LIN {X 0,Y 509.461,Z 538.867,A -85,B 0,C 180,E1 -5497.53,E2 -5497.53} C_VEL
LIN {X 0,Y 509.618,Z 532.772,A -85,B 0,C 180,E1 -5498.525,E2 -5498.525} C_VEL
LIN {X 0,Y 509.848,Z 525.444,A -85,B 0,C 180,E1 -5499.521,E2 -5499.521} C_VEL
LIN {X 0,Y 510.009,Z 518.515,A -85,B 0,C 180,E1 -5500.32,E2 -5500.32} C_VEL
LIN {X 0,Y 510.319,Z 510.334,A -85,B 0,C 180,E1 -5501.116,E2 -5501.116} C_VEL
LIN {X 0,Y 510.583,Z 501.821,A -85,B 0,C 180,E1 -5501.815,E2 -5501.815} C_VEL
LIN {X 0,Y 510.841,Z 492.093,A -85,B 0,C 180,E1 -5502.475,E2 -5502.475} C_VEL
LIN {X 0,Y 511.112,Z 482.332,A -85,B 0,C 180,E1 -5503.012,E2 -5503.012} C_VEL
LIN {X 0,Y 511.344,Z 473.256,A -85,B 0,C 180,E1 -5503.411,E2 -5503.411} C_VEL
LIN {X 0,Y 511.519,Z 463.74,A -85,B 0,C 180,E1 -5503.735,E2 -5503.735} C_VEL
LIN {X 0,Y 511.764,Z 453.432,A -85,B 0,C 180,E1 -5503.981,E2 -5503.981} C_VEL
LIN {X 0,Y 512.128,Z 381.828,A -85,B 0,C 180,E1 -5505.012,E2 -5505.012} C_VEL
LIN {X 0,Y 512.114,Z 359.712,A -85,B 0,C 180,E1 -5505.327,E2 -5505.327} C_VEL
LIN {X 0,Y 510.045,Z 347.334,A -85,B 0,C 180,E1 -5505.59,E2 -5505.59} C_VEL
LIN {X 0,Y 510.232,Z 339.032,A -85,B 0,C 180,E1 -5507.226,E2 -5507.226} C_VEL
LIN {X 0,Y 510.588,Z 324.426,A -85,B 0,C 180,E1 -5510.127,E2 -5510.127} C_VEL
LIN {X 0,Y 510.987,Z 310.909,A -85,B 0,C 180,E1 -5512.852,E2 -5512.852} C_VEL
LIN {X 0,Y 511.208,Z 302.536,A -85,B 0,C 180,E1 -5514.592,E2 -5514.592} C_VEL
LIN {X 0,Y 509.916,Z 294.495,A -85,B 0,C 180,E1 -5516.407,E2 -5516.407} C_VEL
LIN {X 0,Y 509.872,Z 294.473,A -85,B 0,C 180,E1 -5518.844,E2 -5518.844} C_VEL
LIN {X 0,Y 509.82,Z 294.481,A -85,B 0,C 180,E1 -5521.589,E2 -5521.589} C_VEL
LIN {X 0,Y 509.845,Z 294.474,A -85,B 0,C 180,E1 -5524.413,E2 -5524.413} C_VEL
LIN {X 0,Y 509.806,Z 294.478,A -85,B 0,C 180,E1 -5527.341,E2 -5527.341} C_VEL
LIN {X 0,Y 509.835,Z 294.468,A -85,B 0,C 180,E1 -5530.381,E2 -5530.381} C_VEL
LIN {X 0,Y 509.819,Z 294.476,A -85,B 0,C 180,E1 -5533.061,E2 -5533.061} C_VEL
LIN {X 0,Y 509.818,Z 294.48,A -85,B 0,C 180,E1 -5535.792,E2 -5535.792} C_VEL
LIN {X 0,Y 509.854,Z 294.47,A -85,B 0,C 180,E1 -5538.574,E2 -5538.574} C_VEL
LIN {X 0,Y 509.845,Z 294.479,A -85,B 0,C 180,E1 -5541.786,E2 -5541.786} C_VEL
LIN {X 0,Y 509.824,Z 294.472,A -85,B 0,C 180,E1 -5544.621,E2 -5544.621} C_VEL
LIN {X 0,Y 509.853,Z 294.472,A -85,B 0,C 180,E1 -5547.48,E2 -5547.48} C_VEL
LIN {X 0,Y 509.852,Z 294.471,A -85,B 0,C 180,E1 -5550.273,E2 -5550.273} C_VEL
LIN {X 0,Y 509.878,Z 294.462,A -85,B 0,C 180,E1 -5552.944,E2 -5552.944} C_VEL
LIN {X 0,Y 509.839,Z 294.478,A -85,B 0,C 180,E1 -5555.572,E2 -5555.572} C_VEL
LIN {X 0,Y 509.814,Z 294.475,A -85,B 0,C 180,E1 -5558.148,E2 -5558.148} C_VEL
LIN {X 0,Y 509.856,Z 294.463,A -85,B 0,C 180,E1 -5560.681,E2 -5560.681} C_VEL
LIN {X 0,Y 509.876,Z 294.465,A -85,B 0,C 180,E1 -5563.174,E2 -5563.174} C_VEL
LIN {X 0,Y 509.865,Z 294.474,A -85,B 0,C 180,E1 -5565.634,E2 -5565.634} C_VEL
LIN {X 0,Y 509.908,Z 294.462,A -85,B 0,C 180,E1 -5568.874,E2 -5568.874} C_VEL
LIN {X 0,Y 509.943,Z 294.455,A -85,B 0,C 180,E1 -5572.078,E2 -5572.078} C_VEL
LIN {X 0,Y 509.973,Z 294.455,A -85,B 0,C 180,E1 -5574.464,E2 -5574.464} C_VEL
LIN {X 0,Y 510.043,Z 294.446,A -85,B 0,C 180,E1 -5577.63,E2 -5577.63} C_VEL
LIN {X 0,Y 510.043,Z 294.435,A -85,B 0,C 180,E1 -5580,E2 -5580} C_VEL
LIN {X 0,Y 510.044,Z 294.442,A -85,B 0,C 180,E1 -5582.369,E2 -5582.369} C_VEL
LIN {X 0,Y 509.967,Z 294.456,A -85,B 0,C 180,E1 -5586.329,E2 -5586.329} C_VEL
LIN {X 0,Y 509.906,Z 294.463,A -85,B 0,C 180,E1 -5588.72,E2 -5588.72} C_VEL
LIN {X 0,Y 509.895,Z 294.462,A -85,B 0,C 180,E1 -5591.931,E2 -5591.931} C_VEL
LIN {X 0,Y 509.883,Z 294.472,A -85,B 0,C 180,E1 -5595.242,E2 -5595.242} C_VEL
LIN {X 0,Y 509.877,Z 294.462,A -85,B 0,C 180,E1 -5598.001,E2 -5598.001} C_VEL
LIN {X 0,Y 509.84,Z 294.475,A -85,B 0,C 180,E1 -5601.002,E2 -5601.002} C_VEL
LIN {X 0,Y 509.859,Z 294.473,A -85,B 0,C 180,E1 -5604.426,E2 -5604.426} C_VEL
LIN {X 0,Y 509.875,Z 294.466,A -85,B 0,C 180,E1 -5607.056,E2 -5607.056} C_VEL
LIN {X 0,Y 509.871,Z 294.468,A -85,B 0,C 180,E1 -5609.75,E2 -5609.75} C_VEL
LIN {X 0,Y 509.867,Z 294.474,A -85,B 0,C 180,E1 -5612.775,E2 -5612.775} C_VEL
LIN {X 0,Y 509.833,Z 294.471,A -85,B 0,C 180,E1 -5615.581,E2 -5615.581} C_VEL
LIN {X 0,Y 509.843,Z 294.477,A -85,B 0,C 180,E1 -5618.338,E2 -5618.338} C_VEL
LIN {X 0,Y 509.856,Z 294.469,A -85,B 0,C 180,E1 -5621.425,E2 -5621.425} C_VEL
LIN {X 0,Y 509.848,Z 294.476,A -85,B 0,C 180,E1 -5624.668,E2 -5624.668} C_VEL
LIN {X 0,Y 509.853,Z 294.459,A -85,B 0,C 180,E1 -5628.103,E2 -5628.103} C_VEL
LIN {X 0,Y 509.84,Z 294.478,A -85,B 0,C 180,E1 -5630.648,E2 -5630.648} C_VEL
LIN {X 0,Y 509.824,Z 294.473,A -85,B 0,C 180,E1 -5633.749,E2 -5633.749} C_VEL
LIN {X 0,Y 509.159,Z 294.557,A -85,B 0,C 180,E1 -5634.409,E2 -5634.409} C_VEL
LIN {X 0,Y 506.341,Z 294.908,A -85,B 0,C 180,E1 -5635.481,E2 -5635.481} C_VEL
LIN {X 0,Y 503.947,Z 295.208,A -85,B 0,C 180,E1 -5636.344,E2 -5636.344} C_VEL
LIN {X 0,Y 502.899,Z 295.34,A -85,B 0,C 180,E1 -5637.011,E2 -5637.011} C_VEL
LIN {X 0,Y 502.802,Z 295.35,A -85,B 0,C 180,E1 -5637.236,E2 -5637.236} C_VEL
LIN {X 0,Y 502.809,Z 295.351,A -85,B 0,C 180,E1 -5640.065,E2 -5640.065} C_VEL
LIN {X 0,Y 502.83,Z 295.353,A -85,B 0,C 180,E1 -5642.534,E2 -5642.534} C_VEL
LIN {X 0,Y 502.824,Z 295.348,A -85,B 0,C 180,E1 -5645.299,E2 -5645.299} C_VEL
LIN {X 0,Y 502.78,Z 295.356,A -85,B 0,C 180,E1 -5647.827,E2 -5647.827} C_VEL
LIN {X 0,Y 502.822,Z 295.355,A -85,B 0,C 180,E1 -5650.401,E2 -5650.401} C_VEL
LIN {X 0,Y 502.831,Z 295.349,A -85,B 0,C 180,E1 -5652.932,E2 -5652.932} C_VEL
LIN {X 0,Y 502.841,Z 295.347,A -85,B 0,C 180,E1 -5655.429,E2 -5655.429} C_VEL
LIN {X 0,Y 502.874,Z 295.345,A -85,B 0,C 180,E1 -5658.717,E2 -5658.717} C_VEL
LIN {X 0,Y 502.898,Z 295.345,A -85,B 0,C 180,E1 -5661.967,E2 -5661.967} C_VEL
LIN {X 0,Y 502.936,Z 295.339,A -85,B 0,C 180,E1 -5664.387,E2 -5664.387} C_VEL
LIN {X 0,Y 503.023,Z 295.327,A -85,B 0,C 180,E1 -5667.598,E2 -5667.598} C_VEL
LIN {X 0,Y 503.025,Z 295.33,A -85,B 0,C 180,E1 -5670,E2 -5670} C_VEL
LIN {X 0,Y 503.023,Z 295.327,A -85,B 0,C 180,E1 -5672.402,E2 -5672.402} C_VEL
LIN {X 0,Y 502.936,Z 295.339,A -85,B 0,C 180,E1 -5675.613,E2 -5675.613} C_VEL
LIN {X 0,Y 502.898,Z 295.345,A -85,B 0,C 180,E1 -5678.033,E2 -5678.033} C_VEL
LIN {X 0,Y 502.874,Z 295.345,A -85,B 0,C 180,E1 -5681.283,E2 -5681.283} C_VEL
LIN {X 0,Y 502.841,Z 295.347,A -85,B 0,C 180,E1 -5684.571,E2 -5684.571} C_VEL
LIN {X 0,Y 502.858,Z 295.35,A -85,B 0,C 180,E1 -5687.907,E2 -5687.907} C_VEL
LIN {X 0,Y 502.824,Z 295.349,A -85,B 0,C 180,E1 -5690.536,E2 -5690.536} C_VEL
LIN {X 0,Y 502.792,Z 295.354,A -85,B 0,C 180,E1 -5693.04,E2 -5693.04} C_VEL
LIN {X 0,Y 502.837,Z 295.353,A -85,B 0,C 180,E1 -5695.675,E2 -5695.675} C_VEL
LIN {X 0,Y 502.835,Z 295.343,A -85,B 0,C 180,E1 -5698.372,E2 -5698.372} C_VEL
LIN {X 0,Y 502.791,Z 295.358,A -85,B 0,C 180,E1 -5701.499,E2 -5701.499} C_VEL
LIN {X 0,Y 502.8,Z 295.339,A -85,B 0,C 180,E1 -5704.444,E2 -5704.444} C_VEL
LIN {X 0,Y 502.774,Z 295.356,A -85,B 0,C 180,E1 -5707.178,E2 -5707.178} C_VEL
LIN {X 0,Y 502.781,Z 295.347,A -85,B 0,C 180,E1 -5710.015,E2 -5710.015} C_VEL
LIN {X 0,Y 502.795,Z 295.335,A -85,B 0,C 180,E1 -5712.199,E2 -5712.199} C_VEL
LIN {X 0,Y 502.792,Z 295.357,A -85,B 0,C 180,E1 -5715.468,E2 -5715.468} C_VEL
LIN {X 0,Y 502.821,Z 295.347,A -85,B 0,C 180,E1 -5717.864,E2 -5717.864} C_VEL
LIN {X 0,Y 502.801,Z 295.352,A -85,B 0,C 180,E1 -5721.025,E2 -5721.025} C_VEL
LIN {X 0,Y 502.776,Z 295.35,A -85,B 0,C 180,E1 -5724.167,E2 -5724.167} C_VEL
LIN {X 0,Y 502.823,Z 295.348,A -85,B 0,C 180,E1 -5726.993,E2 -5726.993} C_VEL
LIN {X 0,Y 502.821,Z 295.346,A -85,B 0,C 180,E1 -5730.062,E2 -5730.062} C_VEL
LIN {X 0,Y 502.824,Z 295.34,A -85,B 0,C 180,E1 -5732.533,E2 -5732.533} C_VEL
LIN {X 0,Y 502.818,Z 295.353,A -85,B 0,C 180,E1 -5735.298,E2 -5735.298} C_VEL
LIN {X 0,Y 502.783,Z 295.351,A -85,B 0,C 180,E1 -5737.827,E2 -5737.827} C_VEL
LIN {X 0,Y 502.815,Z 295.341,A -85,B 0,C 180,E1 -5740.4,E2 -5740.4} C_VEL
LIN {X 0,Y 502.826,Z 295.348,A -85,B 0,C 180,E1 -5742.932,E2 -5742.932} C_VEL
LIN {X 0,Y 502.834,Z 295.348,A -85,B 0,C 180,E1 -5745.429,E2 -5745.429} C_VEL
LIN {X 0,Y 502.871,Z 295.341,A -85,B 0,C 180,E1 -5748.717,E2 -5748.717} C_VEL
LIN {X 0,Y 502.891,Z 295.333,A -85,B 0,C 180,E1 -5751.967,E2 -5751.967} C_VEL
LIN {X 0,Y 502.928,Z 295.336,A -85,B 0,C 180,E1 -5754.387,E2 -5754.387} C_VEL
LIN {X 0,Y 503.014,Z 295.318,A -85,B 0,C 180,E1 -5757.598,E2 -5757.598} C_VEL
LIN {X 0,Y 503.014,Z 295.309,A -85,B 0,C 180,E1 -5760,E2 -5760} C_VEL
LIN {X 0,Y 503.013,Z 295.322,A -85,B 0,C 180,E1 -5762.403,E2 -5762.403} C_VEL
LIN {X 0,Y 502.929,Z 295.333,A -85,B 0,C 180,E1 -5765.614,E2 -5765.614} C_VEL
LIN {X 0,Y 502.893,Z 295.334,A -85,B 0,C 180,E1 -5768.034,E2 -5768.034} C_VEL
LIN {X 0,Y 502.872,Z 295.337,A -85,B 0,C 180,E1 -5771.284,E2 -5771.284} C_VEL
LIN {X 0,Y 502.843,Z 295.351,A -85,B 0,C 180,E1 -5774.571,E2 -5774.571} C_VEL
LIN {X 0,Y 502.853,Z 295.336,A -85,B 0,C 180,E1 -5777.908,E2 -5777.908} C_VEL
LIN {X 0,Y 502.821,Z 295.349,A -85,B 0,C 180,E1 -5780.537,E2 -5780.537} C_VEL
LIN {X 0,Y 502.781,Z 295.353,A -85,B 0,C 180,E1 -5783.042,E2 -5783.042} C_VEL
LIN {X 0,Y 502.814,Z 295.343,A -85,B 0,C 180,E1 -5785.677,E2 -5785.677} C_VEL
LIN {X 0,Y 502.834,Z 295.347,A -85,B 0,C 180,E1 -5788.373,E2 -5788.373} C_VEL
LIN {X 0,Y 502.786,Z 295.351,A -85,B 0,C 180,E1 -5791.5,E2 -5791.5} C_VEL
LIN {X 0,Y 502.785,Z 295.353,A -85,B 0,C 180,E1 -5794.443,E2 -5794.443} C_VEL
LIN {X 0,Y 502.772,Z 295.353,A -85,B 0,C 180,E1 -5797.179,E2 -5797.179} C_VEL
LIN {X 0,Y 502.783,Z 295.354,A -85,B 0,C 180,E1 -5800.016,E2 -5800.016} C_VEL
LIN {X 0,Y 502.799,Z 295.358,A -85,B 0,C 180,E1 -5802.2,E2 -5802.2} C_VEL
LIN {X 0,Y 502.782,Z 295.352,A -85,B 0,C 180,E1 -5805.471,E2 -5805.471} C_VEL
LIN {X 0,Y 502.792,Z 295.356,A -85,B 0,C 180,E1 -5807.861,E2 -5807.861} C_VEL
LIN {X 0,Y 502.798,Z 295.349,A -85,B 0,C 180,E1 -5811.025,E2 -5811.025} C_VEL
LIN {X 0,Y 502.769,Z 295.354,A -85,B 0,C 180,E1 -5814.171,E2 -5814.171} C_VEL
LIN {X 0,Y 502.832,Z 295.345,A -85,B 0,C 180,E1 -5816.994,E2 -5816.994} C_VEL
LIN {X 0,Y 502.815,Z 295.352,A -85,B 0,C 180,E1 -5820.066,E2 -5820.066} C_VEL
LIN {X 0,Y 502.868,Z 295.346,A -85,B 0,C 180,E1 -5823.211,E2 -5823.211} C_VEL
LIN {X 0,Y 502.924,Z 295.7,A -85,B 0,C 180,E1 -5823.524,E2 -5823.524} C_VEL
LIN {X 0,Y 504.235,Z 303.512,A -85,B 0,C 180,E1 -5825.284,E2 -5825.284} C_VEL
LIN {X 0,Y 503.886,Z 315.919,A -85,B 0,C 180,E1 -5827.878,E2 -5827.878} C_VEL
LIN {X 0,Y 503.426,Z 330.518,A -85,B 0,C 180,E1 -5830.849,E2 -5830.849} C_VEL
LIN {X 0,Y 503.056,Z 344.925,A -85,B 0,C 180,E1 -5833.775,E2 -5833.775} C_VEL
LIN {X 0,Y 503.018,Z 347.127,A -85,B 0,C 180,E1 -5834.185,E2 -5834.185} C_VEL
LIN {X 0,Y 505.389,Z 362.648,A -85,B 0,C 180,E1 -5834.509,E2 -5834.509} C_VEL
LIN {X 0,Y 504.882,Z 451.906,A -85,B 0,C 180,E1 -5835.798,E2 -5835.798} C_VEL
LIN {X 0,Y 504.667,Z 462.672,A -85,B 0,C 180,E1 -5836.049,E2 -5836.049} C_VEL
LIN {X 0,Y 504.48,Z 471.774,A -85,B 0,C 180,E1 -5836.352,E2 -5836.352} C_VEL
LIN {X 0,Y 504.159,Z 482.137,A -85,B 0,C 180,E1 -5836.805,E2 -5836.805} C_VEL
LIN {X 0,Y 503.896,Z 492.03,A -85,B 0,C 180,E1 -5837.358,E2 -5837.358} C_VEL
LIN {X 0,Y 503.667,Z 500.274,A -85,B 0,C 180,E1 -5837.919,E2 -5837.919} C_VEL
LIN {X 0,Y 503.36,Z 509.004,A -85,B 0,C 180,E1 -5838.626,E2 -5838.626} C_VEL
LIN {X 0,Y 503.083,Z 516.401,A -85,B 0,C 180,E1 -5839.333,E2 -5839.333} C_VEL
LIN {X 0,Y 502.851,Z 523.622,A -85,B 0,C 180,E1 -5840.142,E2 -5840.142} C_VEL
LIN {X 0,Y 502.652,Z 529.825,A -85,B 0,C 180,E1 -5840.95,E2 -5840.95} C_VEL
LIN {X 0,Y 502.478,Z 536.362,A -85,B 0,C 180,E1 -5841.96,E2 -5841.96} C_VEL
LIN {X 0,Y 502.328,Z 541.916,A -85,B 0,C 180,E1 -5842.989,E2 -5842.989} C_VEL
LIN {X 0,Y 502.208,Z 546.351,A -85,B 0,C 180,E1 -5843.975,E2 -5843.975} C_VEL
LIN {X 0,Y 502.114,Z 550.671,A -85,B 0,C 180,E1 -5845.183,E2 -5845.183} C_VEL
LIN {X 0,Y 502.139,Z 553.036,A -85,B 0,C 180,E1 -5845.987,E2 -5845.987} C_VEL
LIN {X 0,Y 502.12,Z 554.831,A -85,B 0,C 180,E1 -5846.791,E2 -5846.791} C_VEL
LIN {X 0,Y 502.037,Z 557.269,A -85,B 0,C 180,E1 -5848.396,E2 -5848.396} C_VEL
LIN {X 0,Y 501.991,Z 557.855,A -85,B 0,C 180,E1 -5849.198,E2 -5849.198} C_VEL
LIN {X 0,Y 501.991,Z 557.855,A -85,B 0,C 180,E1 -5850.802,E2 -5850.802} C_VEL
LIN {X 0,Y 502.037,Z 557.269,A -85,B 0,C 180,E1 -5851.604,E2 -5851.604} C_VEL
LIN {X 0,Y 502.12,Z 554.831,A -85,B 0,C 180,E1 -5853.209,E2 -5853.209} C_VEL
LIN {X 0,Y 502.105,Z 551.886,A -85,B 0,C 180,E1 -5854.415,E2 -5854.415} C_VEL
LIN {X 0,Y 502.205,Z 547.904,A -85,B 0,C 180,E1 -5855.622,E2 -5855.622} C_VEL
LIN {X 0,Y 502.27,Z 542.969,A -85,B 0,C 180,E1 -5856.79,E2 -5856.79} C_VEL
LIN {X 0,Y 502.409,Z 537.517,A -85,B 0,C 180,E1 -5857.839,E2 -5857.839} C_VEL
LIN {X 0,Y 502.597,Z 531.2,A -85,B 0,C 180,E1 -5858.848,E2 -5858.848} C_VEL
LIN {X 0,Y 502.807,Z 525.249,A -85,B 0,C 180,E1 -5859.656,E2 -5859.656} C_VEL
LIN {X 0,Y 502.987,Z 518.32,A -85,B 0,C 180,E1 -5860.465,E2 -5860.465} C_VEL
LIN {X 0,Y 503.306,Z 510.139,A -85,B 0,C 180,E1 -5861.273,E2 -5861.273} C_VEL
LIN {X 0,Y 503.602,Z 501.626,A -85,B 0,C 180,E1 -5861.981,E2 -5861.981} C_VEL
LIN {X 0,Y 503.872,Z 492.358,A -85,B 0,C 180,E1 -5862.622,E2 -5862.622} C_VEL
LIN {X 0,Y 504.155,Z 483.145,A -85,B 0,C 180,E1 -5863.144,E2 -5863.144} C_VEL
LIN {X 0,Y 504.445,Z 473.062,A -85,B 0,C 180,E1 -5863.597,E2 -5863.597} C_VEL
LIN {X 0,Y 504.639,Z 463.546,A -85,B 0,C 180,E1 -5863.926,E2 -5863.926} C_VEL
LIN {X 0,Y 504.869,Z 453.238,A -85,B 0,C 180,E1 -5864.176,E2 -5864.176} C_VEL
LIN {X 0,Y 505.244,Z 390.584,A -85,B 0,C 180,E1 -5865.092,E2 -5865.092} C_VEL
LIN {X 0,Y 505.248,Z 360.522,A -85,B 0,C 180,E1 -5865.526,E2 -5865.526} C_VEL
LIN {X 0,Y 503.065,Z 347.271,A -85,B 0,C 180,E1 -5865.804,E2 -5865.804} C_VEL
LIN {X 0,Y 503.028,Z 346.232,A -85,B 0,C 180,E1 -5865.944,E2 -5865.944} C_VEL
LIN {X 0,Y 503.374,Z 332.655,A -85,B 0,C 180,E1 -5868.73,E2 -5868.73} C_VEL
LIN {X 0,Y 503.873,Z 316.967,A -85,B 0,C 180,E1 -5871.907,E2 -5871.907} C_VEL
LIN {X 0,Y 504.263,Z 304.576,A -85,B 0,C 180,E1 -5874.495,E2 -5874.495} C_VEL
LIN {X 0,Y 503.045,Z 296.318,A -85,B 0,C 180,E1 -5876.332,E2 -5876.332} C_VEL
LIN {X 0,Y 502.855,Z 295.361,A -85,B 0,C 180,E1 -5876.622,E2 -5876.622} C_VEL
LIN {X 0,Y 502.822,Z 295.351,A -85,B 0,C 180,E1 -5879.287,E2 -5879.287} C_VEL
LIN {X 0,Y 502.783,Z 295.355,A -85,B 0,C 180,E1 -5882.084,E2 -5882.084} C_VEL
LIN {X 0,Y 502.796,Z 295.35,A -85,B 0,C 180,E1 -5884.965,E2 -5884.965} C_VEL
LIN {X 0,Y 502.791,Z 295.352,A -85,B 0,C 180,E1 -5888.485,E2 -5888.485} C_VEL
LIN {X 0,Y 502.798,Z 295.342,A -85,B 0,C 180,E1 -5891.067,E2 -5891.067} C_VEL
LIN {X 0,Y 502.775,Z 295.354,A -85,B 0,C 180,E1 -5894.339,E2 -5894.339} C_VEL
LIN {X 0,Y 502.768,Z 295.353,A -85,B 0,C 180,E1 -5896.768,E2 -5896.768} C_VEL
LIN {X 0,Y 502.815,Z 295.347,A -85,B 0,C 180,E1 -5899.004,E2 -5899.004} C_VEL
LIN {X 0,Y 502.788,Z 295.356,A -85,B 0,C 180,E1 -5902.045,E2 -5902.045} C_VEL
LIN {X 0,Y 502.79,Z 295.349,A -85,B 0,C 180,E1 -5905.033,E2 -5905.033} C_VEL
LIN {X 0,Y 502.776,Z 295.357,A -85,B 0,C 180,E1 -5907.914,E2 -5907.914} C_VEL
LIN {X 0,Y 502.817,Z 295.346,A -85,B 0,C 180,E1 -5910.711,E2 -5910.711} C_VEL
LIN {X 0,Y 502.855,Z 295.34,A -85,B 0,C 180,E1 -5913.438,E2 -5913.438} C_VEL
LIN {X 0,Y 502.766,Z 295.355,A -85,B 0,C 180,E1 -5916.085,E2 -5916.085} C_VEL
LIN {X 0,Y 502.775,Z 295.351,A -85,B 0,C 180,E1 -5918.688,E2 -5918.688} C_VEL
LIN {X 0,Y 502.822,Z 295.343,A -85,B 0,C 180,E1 -5921.248,E2 -5921.248} C_VEL
LIN {X 0,Y 502.814,Z 295.35,A -85,B 0,C 180,E1 -5923.766,E2 -5923.766} C_VEL
LIN {X 0,Y 502.827,Z 295.345,A -85,B 0,C 180,E1 -5926.254,E2 -5926.254} C_VEL
LIN {X 0,Y 502.872,Z 295.337,A -85,B 0,C 180,E1 -5928.716,E2 -5928.716} C_VEL
LIN {X 0,Y 502.893,Z 295.334,A -85,B 0,C 180,E1 -5931.966,E2 -5931.966} C_VEL
LIN {X 0,Y 502.929,Z 295.333,A -85,B 0,C 180,E1 -5934.386,E2 -5934.386} C_VEL
LIN {X 0,Y 503.013,Z 295.322,A -85,B 0,C 180,E1 -5937.597,E2 -5937.597} C_VEL
LIN {X 0,Y 503.014,Z 295.309,A -85,B 0,C 180,E1 -5940,E2 -5940} C_VEL
LIN {X 0,Y 503.014,Z 295.318,A -85,B 0,C 180,E1 -5942.402,E2 -5942.402} C_VEL
LIN {X 0,Y 502.929,Z 295.336,A -85,B 0,C 180,E1 -5945.613,E2 -5945.613} C_VEL
LIN {X 0,Y 502.891,Z 295.333,A -85,B 0,C 180,E1 -5948.033,E2 -5948.033} C_VEL
LIN {X 0,Y 502.871,Z 295.341,A -85,B 0,C 180,E1 -5951.283,E2 -5951.283} C_VEL
LIN {X 0,Y 502.834,Z 295.348,A -85,B 0,C 180,E1 -5954.571,E2 -5954.571} C_VEL
LIN {X 0,Y 502.851,Z 295.337,A -85,B 0,C 180,E1 -5957.907,E2 -5957.907} C_VEL
LIN {X 0,Y 502.818,Z 295.342,A -85,B 0,C 180,E1 -5960.536,E2 -5960.536} C_VEL
LIN {X 0,Y 502.783,Z 295.359,A -85,B 0,C 180,E1 -5963.04,E2 -5963.04} C_VEL
LIN {X 0,Y 502.83,Z 295.342,A -85,B 0,C 180,E1 -5965.676,E2 -5965.676} C_VEL
LIN {X 0,Y 502.832,Z 295.341,A -85,B 0,C 180,E1 -5968.373,E2 -5968.373} C_VEL
LIN {X 0,Y 502.787,Z 295.352,A -85,B 0,C 180,E1 -5971.5,E2 -5971.5} C_VEL
LIN {X 0,Y 502.798,Z 295.35,A -85,B 0,C 180,E1 -5974.445,E2 -5974.445} C_VEL
LIN {X 0,Y 502.772,Z 295.356,A -85,B 0,C 180,E1 -5977.179,E2 -5977.179} C_VEL
LIN {X 0,Y 502.813,Z 295.347,A -85,B 0,C 180,E1 -5980.012,E2 -5980.012} C_VEL
LIN {X 0,Y 502.821,Z 295.347,A -85,B 0,C 180,E1 -5982.203,E2 -5982.203} C_VEL
LIN {X 0,Y 502.792,Z 295.346,A -85,B 0,C 180,E1 -5985.469,E2 -5985.469} C_VEL
LIN {X 0,Y 502.822,Z 295.332,A -85,B 0,C 180,E1 -5987.865,E2 -5987.865} C_VEL
LIN {X 0,Y 502.795,Z 295.353,A -85,B 0,C 180,E1 -5991.024,E2 -5991.024} C_VEL
LIN {X 0,Y 502.779,Z 295.355,A -85,B 0,C 180,E1 -5994.167,E2 -5994.167} C_VEL
LIN {X 0,Y 502.802,Z 295.35,A -85,B 0,C 180,E1 -5997.236,E2 -5997.236} C_VEL
LIN {X 0,Y 502.103,Z 295.44,A -85,B 0,C 180,E1 -5997.905,E2 -5997.905} C_VEL
LIN {X 0,Y 499.238,Z 295.794,A -85,B 0,C 180,E1 -5998.991,E2 -5998.991} C_VEL
LIN {X 0,Y 496.842,Z 296.093,A -85,B 0,C 180,E1 -5999.866,E2 -5999.866} C_VEL
LIN {X 0,Y 495.825,Z 296.217,A -85,B 0,C 180,E1 -6000.541,E2 -6000.541} C_VEL
LIN {X 0,Y 495.747,Z 296.225,A -85,B 0,C 180,E1 -6000.77,E2 -6000.77} C_VEL
LIN {X 0,Y 495.794,Z 296.227,A -85,B 0,C 180,E1 -6003.933,E2 -6003.933} C_VEL
LIN {X 0,Y 495.76,Z 296.229,A -85,B 0,C 180,E1 -6007.138,E2 -6007.138} C_VEL
LIN {X 0,Y 495.768,Z 296.233,A -85,B 0,C 180,E1 -6010.11,E2 -6010.11} C_VEL
LIN {X 0,Y 495.784,Z 296.229,A -85,B 0,C 180,E1 -6012.682,E2 -6012.682} C_VEL
LIN {X 0,Y 495.786,Z 296.226,A -85,B 0,C 180,E1 -6015.217,E2 -6015.217} C_VEL
LIN {X 0,Y 495.848,Z 296.222,A -85,B 0,C 180,E1 -6018.555,E2 -6018.555} C_VEL
LIN {X 0,Y 495.869,Z 296.22,A -85,B 0,C 180,E1 -6021.852,E2 -6021.852} C_VEL
LIN {X 0,Y 495.893,Z 296.217,A -85,B 0,C 180,E1 -6024.307,E2 -6024.307} C_VEL
LIN {X 0,Y 495.991,Z 296.203,A -85,B 0,C 180,E1 -6027.564,E2 -6027.564} C_VEL
LIN {X 0,Y 495.996,Z 296.206,A -85,B 0,C 180,E1 -6030,E2 -6030} C_VEL
LIN {X 0,Y 495.991,Z 296.203,A -85,B 0,C 180,E1 -6032.436,E2 -6032.436} C_VEL
LIN {X 0,Y 495.893,Z 296.217,A -85,B 0,C 180,E1 -6035.693,E2 -6035.693} C_VEL
LIN {X 0,Y 495.869,Z 296.22,A -85,B 0,C 180,E1 -6038.148,E2 -6038.148} C_VEL
LIN {X 0,Y 495.848,Z 296.222,A -85,B 0,C 180,E1 -6041.445,E2 -6041.445} C_VEL
LIN {X 0,Y 495.786,Z 296.226,A -85,B 0,C 180,E1 -6044.783,E2 -6044.783} C_VEL
LIN {X 0,Y 495.784,Z 296.229,A -85,B 0,C 180,E1 -6047.318,E2 -6047.318} C_VEL
LIN {X 0,Y 495.768,Z 296.233,A -85,B 0,C 180,E1 -6049.89,E2 -6049.89} C_VEL
LIN {X 0,Y 495.76,Z 296.229,A -85,B 0,C 180,E1 -6052.862,E2 -6052.862} C_VEL
LIN {X 0,Y 495.794,Z 296.227,A -85,B 0,C 180,E1 -6056.067,E2 -6056.067} C_VEL
LIN {X 0,Y 495.766,Z 296.223,A -85,B 0,C 180,E1 -6058.814,E2 -6058.814} C_VEL
LIN {X 0,Y 495.753,Z 296.234,A -85,B 0,C 180,E1 -6061.726,E2 -6061.726} C_VEL
LIN {X 0,Y 495.77,Z 296.214,A -85,B 0,C 180,E1 -6064.695,E2 -6064.695} C_VEL
LIN {X 0,Y 495.725,Z 296.24,A -85,B 0,C 180,E1 -6067.561,E2 -6067.561} C_VEL
LIN {X 0,Y 495.759,Z 296.22,A -85,B 0,C 180,E1 -6070.699,E2 -6070.699} C_VEL
LIN {X 0,Y 495.726,Z 296.229,A -85,B 0,C 180,E1 -6073.695,E2 -6073.695} C_VEL
LIN {X 0,Y 495.72,Z 296.232,A -85,B 0,C 180,E1 -6076.305,E2 -6076.305} C_VEL
LIN {X 0,Y 495.771,Z 296.227,A -85,B 0,C 180,E1 -6079.301,E2 -6079.301} C_VEL
LIN {X 0,Y 495.722,Z 296.232,A -85,B 0,C 180,E1 -6082.438,E2 -6082.438} C_VEL
LIN {X 0,Y 495.776,Z 296.224,A -85,B 0,C 180,E1 -6085.457,E2 -6085.457} C_VEL
LIN {X 0,Y 495.749,Z 296.228,A -85,B 0,C 180,E1 -6088.364,E2 -6088.364} C_VEL
LIN {X 0,Y 495.78,Z 296.22,A -85,B 0,C 180,E1 -6091.506,E2 -6091.506} C_VEL
LIN {X 0,Y 495.78,Z 296.22,A -85,B 0,C 180,E1 -6093.932,E2 -6093.932} C_VEL
LIN {X 0,Y 495.747,Z 296.235,A -85,B 0,C 180,E1 -6097.14,E2 -6097.14} C_VEL
LIN {X 0,Y 495.767,Z 296.217,A -85,B 0,C 180,E1 -6100.11,E2 -6100.11} C_VEL
LIN {X 0,Y 495.777,Z 296.221,A -85,B 0,C 180,E1 -6102.682,E2 -6102.682} C_VEL
LIN {X 0,Y 495.779,Z 296.229,A -85,B 0,C 180,E1 -6105.217,E2 -6105.217} C_VEL
LIN {X 0,Y 495.844,Z 296.215,A -85,B 0,C 180,E1 -6108.555,E2 -6108.555} C_VEL
LIN {X 0,Y 495.863,Z 296.208,A -85,B 0,C 180,E1 -6111.852,E2 -6111.852} C_VEL
LIN {X 0,Y 495.886,Z 296.212,A -85,B 0,C 180,E1 -6114.307,E2 -6114.307} C_VEL
LIN {X 0,Y 495.983,Z 296.193,A -85,B 0,C 180,E1 -6117.564,E2 -6117.564} C_VEL
LIN {X 0,Y 495.986,Z 296.184,A -85,B 0,C 180,E1 -6120,E2 -6120} C_VEL
LIN {X 0,Y 495.982,Z 296.198,A -85,B 0,C 180,E1 -6122.437,E2 -6122.437} C_VEL
LIN {X 0,Y 495.886,Z 296.21,A -85,B 0,C 180,E1 -6125.694,E2 -6125.694} C_VEL
LIN {X 0,Y 495.864,Z 296.21,A -85,B 0,C 180,E1 -6128.149,E2 -6128.149} C_VEL
LIN {X 0,Y 495.845,Z 296.211,A -85,B 0,C 180,E1 -6131.446,E2 -6131.446} C_VEL
LIN {X 0,Y 495.786,Z 296.227,A -85,B 0,C 180,E1 -6134.783,E2 -6134.783} C_VEL
LIN {X 0,Y 495.789,Z 296.218,A -85,B 0,C 180,E1 -6138.172,E2 -6138.172} C_VEL
LIN {X 0,Y 495.766,Z 296.229,A -85,B 0,C 180,E1 -6140.757,E2 -6140.757} C_VEL
LIN {X 0,Y 495.735,Z 296.229,A -85,B 0,C 180,E1 -6143.388,E2 -6143.388} C_VEL
LIN {X 0,Y 495.816,Z 296.215,A -85,B 0,C 180,E1 -6146.75,E2 -6146.75} C_VEL
LIN {X 0,Y 495.759,Z 296.227,A -85,B 0,C 180,E1 -6149.747,E2 -6149.747} C_VEL
LIN {X 0,Y 495.745,Z 296.228,A -85,B 0,C 180,E1 -6152.596,E2 -6152.596} C_VEL
LIN {X 0,Y 495.741,Z 296.226,A -85,B 0,C 180,E1 -6155.539,E2 -6155.539} C_VEL
LIN {X 0,Y 495.758,Z 296.226,A -85,B 0,C 180,E1 -6158.769,E2 -6158.769} C_VEL
LIN {X 0,Y 495.753,Z 296.23,A -85,B 0,C 180,E1 -6161.782,E2 -6161.782} C_VEL
LIN {X 0,Y 495.733,Z 296.229,A -85,B 0,C 180,E1 -6165.142,E2 -6165.142} C_VEL
LIN {X 0,Y 495.748,Z 296.227,A -85,B 0,C 180,E1 -6168.219,E2 -6168.219} C_VEL
LIN {X 0,Y 495.747,Z 296.229,A -85,B 0,C 180,E1 -6171.409,E2 -6171.409} C_VEL
LIN {X 0,Y 495.743,Z 296.23,A -85,B 0,C 180,E1 -6174.463,E2 -6174.463} C_VEL
LIN {X 0,Y 495.767,Z 296.227,A -85,B 0,C 180,E1 -6177.406,E2 -6177.406} C_VEL
LIN {X 0,Y 495.766,Z 296.23,A -85,B 0,C 180,E1 -6180.254,E2 -6180.254} C_VEL
LIN {X 0,Y 495.849,Z 296.316,A -85,B 0,C 180,E1 -6183.246,E2 -6183.246} C_VEL
LIN {X 0,Y 497.307,Z 305.46,A -85,B 0,C 180,E1 -6185.362,E2 -6185.362} C_VEL
LIN {X 0,Y 496.819,Z 319.971,A -85,B 0,C 180,E1 -6188.421,E2 -6188.421} C_VEL
LIN {X 0,Y 496.323,Z 335.218,A -85,B 0,C 180,E1 -6191.574,E2 -6191.574} C_VEL
LIN {X 0,Y 496,Z 346.756,A -85,B 0,C 180,E1 -6193.94,E2 -6193.94} C_VEL
LIN {X 0,Y 496.799,Z 351.788,A -85,B 0,C 180,E1 -6194.078,E2 -6194.078} C_VEL
LIN {X 0,Y 498.535,Z 363.439,A -85,B 0,C 180,E1 -6194.305,E2 -6194.305} C_VEL
LIN {X 0,Y 497.999,Z 451.712,A -85,B 0,C 180,E1 -6195.598,E2 -6195.598} C_VEL
LIN {X 0,Y 497.791,Z 462.479,A -85,B 0,C 180,E1 -6195.853,E2 -6195.853} C_VEL
LIN {X 0,Y 497.586,Z 471.58,A -85,B 0,C 180,E1 -6196.159,E2 -6196.159} C_VEL
LIN {X 0,Y 497.238,Z 481.943,A -85,B 0,C 180,E1 -6196.618,E2 -6196.618} C_VEL
LIN {X 0,Y 496.997,Z 490.78,A -85,B 0,C 180,E1 -6197.112,E2 -6197.112} C_VEL
LIN {X 0,Y 496.685,Z 500.079,A -85,B 0,C 180,E1 -6197.746,E2 -6197.746} C_VEL
LIN {X 0,Y 496.387,Z 508.81,A -85,B 0,C 180,E1 -6198.464,E2 -6198.464} C_VEL
LIN {X 0,Y 496.097,Z 516.207,A -85,B 0,C 180,E1 -6199.181,E2 -6199.181} C_VEL
LIN {X 0,Y 495.83,Z 523.427,A -85,B 0,C 180,E1 -6200.001,E2 -6200.001} C_VEL
LIN {X 0,Y 495.619,Z 529.63,A -85,B 0,C 180,E1 -6200.821,E2 -6200.821} C_VEL
LIN {X 0,Y 495.403,Z 536.167,A -85,B 0,C 180,E1 -6201.844,E2 -6201.844} C_VEL
LIN {X 0,Y 495.27,Z 540.668,A -85,B 0,C 180,E1 -6202.663,E2 -6202.663} C_VEL
LIN {X 0,Y 495.122,Z 545.679,A -85,B 0,C 180,E1 -6203.763,E2 -6203.763} C_VEL
LIN {X 0,Y 495.107,Z 549.239,A -85,B 0,C 180,E1 -6204.706,E2 -6204.706} C_VEL
LIN {X 0,Y 495.033,Z 552.841,A -85,B 0,C 180,E1 -6205.93,E2 -6205.93} C_VEL
LIN {X 0,Y 495.042,Z 554.638,A -85,B 0,C 180,E1 -6206.745,E2 -6206.745} C_VEL
LIN {X 0,Y 494.963,Z 557.076,A -85,B 0,C 180,E1 -6208.373,E2 -6208.373} C_VEL
LIN {X 0,Y 494.911,Z 557.662,A -85,B 0,C 180,E1 -6209.186,E2 -6209.186} C_VEL
LIN {X 0,Y 494.911,Z 557.662,A -85,B 0,C 180,E1 -6210.814,E2 -6210.814} C_VEL
LIN {X 0,Y 494.963,Z 557.076,A -85,B 0,C 180,E1 -6211.627,E2 -6211.627} C_VEL
LIN {X 0,Y 495.042,Z 554.638,A -85,B 0,C 180,E1 -6213.255,E2 -6213.255} C_VEL
LIN {X 0,Y 495.011,Z 551.692,A -85,B 0,C 180,E1 -6214.479,E2 -6214.479} C_VEL
LIN {X 0,Y 495.121,Z 547.71,A -85,B 0,C 180,E1 -6215.702,E2 -6215.702} C_VEL
LIN {X 0,Y 495.198,Z 542.582,A -85,B 0,C 180,E1 -6216.929,E2 -6216.929} C_VEL
LIN {X 0,Y 495.361,Z 537.322,A -85,B 0,C 180,E1 -6217.951,E2 -6217.951} C_VEL
LIN {X 0,Y 495.563,Z 531.006,A -85,B 0,C 180,E1 -6218.975,E2 -6218.975} C_VEL
LIN {X 0,Y 495.757,Z 525.054,A -85,B 0,C 180,E1 -6219.794,E2 -6219.794} C_VEL
LIN {X 0,Y 495.985,Z 518.125,A -85,B 0,C 180,E1 -6220.615,E2 -6220.615} C_VEL
LIN {X 0,Y 496.328,Z 509.945,A -85,B 0,C 180,E1 -6221.434,E2 -6221.434} C_VEL
LIN {X 0,Y 496.606,Z 501.43,A -85,B 0,C 180,E1 -6222.152,E2 -6222.152} C_VEL
LIN {X 0,Y 496.909,Z 492.637,A -85,B 0,C 180,E1 -6222.772,E2 -6222.772} C_VEL
LIN {X 0,Y 497.209,Z 482.95,A -85,B 0,C 180,E1 -6223.331,E2 -6223.331} C_VEL
LIN {X 0,Y 497.499,Z 474.156,A -85,B 0,C 180,E1 -6223.739,E2 -6223.739} C_VEL
LIN {X 0,Y 497.739,Z 464.227,A -85,B 0,C 180,E1 -6224.097,E2 -6224.097} C_VEL
LIN {X 0,Y 497.98,Z 454.376,A -85,B 0,C 180,E1 -6224.351,E2 -6224.351} C_VEL
LIN {X 0,Y 498.169,Z 429.799,A -85,B 0,C 180,E1 -6224.736,E2 -6224.736} C_VEL
LIN {X 0,Y 498.489,Z 361.816,A -85,B 0,C 180,E1 -6225.72,E2 -6225.72} C_VEL
LIN {X 0,Y 496.042,Z 347.085,A -85,B 0,C 180,E1 -6226.034,E2 -6226.034} C_VEL
LIN {X 0,Y 496.031,Z 345.706,A -85,B 0,C 180,E1 -6226.25,E2 -6226.25} C_VEL
LIN {X 0,Y 496.434,Z 331.477,A -85,B 0,C 180,E1 -6229.217,E2 -6229.217} C_VEL
LIN {X 0,Y 496.906,Z 317.878,A -85,B 0,C 180,E1 -6232.012,E2 -6232.012} C_VEL
LIN {X 0,Y 497.311,Z 305.5,A -85,B 0,C 180,E1 -6234.638,E2 -6234.638} C_VEL
LIN {X 0,Y 495.832,Z 296.253,A -85,B 0,C 180,E1 -6236.778,E2 -6236.778} C_VEL
LIN {X 0,Y 495.766,Z 296.23,A -85,B 0,C 180,E1 -6239.746,E2 -6239.746} C_VEL
LIN {X 0,Y 495.767,Z 296.227,A -85,B 0,C 180,E1 -6242.594,E2 -6242.594} C_VEL
LIN {X 0,Y 495.743,Z 296.23,A -85,B 0,C 180,E1 -6245.537,E2 -6245.537} C_VEL
LIN {X 0,Y 495.76,Z 296.226,A -85,B 0,C 180,E1 -6248.767,E2 -6248.767} C_VEL
LIN {X 0,Y 495.748,Z 296.227,A -85,B 0,C 180,E1 -6251.781,E2 -6251.781} C_VEL
LIN {X 0,Y 495.733,Z 296.23,A -85,B 0,C 180,E1 -6255.14,E2 -6255.14} C_VEL
LIN {X 0,Y 495.753,Z 296.23,A -85,B 0,C 180,E1 -6258.218,E2 -6258.218} C_VEL
LIN {X 0,Y 495.745,Z 296.229,A -85,B 0,C 180,E1 -6261.407,E2 -6261.407} C_VEL
LIN {X 0,Y 495.741,Z 296.226,A -85,B 0,C 180,E1 -6264.461,E2 -6264.461} C_VEL
LIN {X 0,Y 495.745,Z 296.228,A -85,B 0,C 180,E1 -6267.404,E2 -6267.404} C_VEL
LIN {X 0,Y 495.759,Z 296.227,A -85,B 0,C 180,E1 -6270.253,E2 -6270.253} C_VEL
LIN {X 0,Y 495.816,Z 296.215,A -85,B 0,C 180,E1 -6273.25,E2 -6273.25} C_VEL
LIN {X 0,Y 495.735,Z 296.229,A -85,B 0,C 180,E1 -6276.612,E2 -6276.612} C_VEL
LIN {X 0,Y 495.77,Z 296.229,A -85,B 0,C 180,E1 -6279.323,E2 -6279.323} C_VEL
LIN {X 0,Y 495.789,Z 296.218,A -85,B 0,C 180,E1 -6281.828,E2 -6281.828} C_VEL
LIN {X 0,Y 495.815,Z 296.217,A -85,B 0,C 180,E1 -6284.548,E2 -6284.548} C_VEL
LIN {X 0,Y 495.82,Z 296.216,A -85,B 0,C 180,E1 -6287.964,E2 -6287.964} C_VEL
LIN {X 0,Y 495.836,Z 296.207,A -85,B 0,C 180,E1 -6291.03,E2 -6291.03} C_VEL
LIN {X 0,Y 495.87,Z 296.218,A -85,B 0,C 180,E1 -6293.489,E2 -6293.489} C_VEL
LIN {X 0,Y 495.835,Z 296.219,A -85,B 0,C 180,E1 -6296.749,E2 -6296.749} C_VEL
LIN {X 0,Y 495.997,Z 296.192,A -85,B 0,C 180,E1 -6299.188,E2 -6299.188} C_VEL
LIN {X 0,Y 495.861,Z 296.211,A -85,B 0,C 180,E1 -6301.624,E2 -6301.624} C_VEL
LIN {X 0,Y 495.836,Z 296.222,A -85,B 0,C 180,E1 -6303.25,E2 -6303.25} C_VEL
LIN {X 0,Y 495.869,Z 296.214,A -85,B 0,C 180,E1 -6306.51,E2 -6306.51} C_VEL
LIN {X 0,Y 495.834,Z 296.214,A -85,B 0,C 180,E1 -6308.969,E2 -6308.969} C_VEL
LIN {X 0,Y 495.808,Z 296.216,A -85,B 0,C 180,E1 -6312.276,E2 -6312.276} C_VEL
LIN {X 0,Y 495.797,Z 296.222,A -85,B 0,C 180,E1 -6315.624,E2 -6315.624} C_VEL
LIN {X 0,Y 495.796,Z 296.216,A -85,B 0,C 180,E1 -6318.247,E2 -6318.247} C_VEL
LIN {X 0,Y 495.763,Z 296.224,A -85,B 0,C 180,E1 -6320.756,E2 -6320.756} C_VEL
LIN {X 0,Y 495.741,Z 296.231,A -85,B 0,C 180,E1 -6323.387,E2 -6323.387} C_VEL
LIN {X 0,Y 495.78,Z 296.22,A -85,B 0,C 180,E1 -6326.068,E2 -6326.068} C_VEL
LIN {X 0,Y 495.771,Z 296.226,A -85,B 0,C 180,E1 -6328.814,E2 -6328.814} C_VEL
LIN {X 0,Y 495.749,Z 296.228,A -85,B 0,C 180,E1 -6331.726,E2 -6331.726} C_VEL
LIN {X 0,Y 495.767,Z 296.225,A -85,B 0,C 180,E1 -6334.696,E2 -6334.696} C_VEL
LIN {X 0,Y 495.722,Z 296.232,A -85,B 0,C 180,E1 -6337.562,E2 -6337.562} C_VEL
LIN {X 0,Y 495.771,Z 296.227,A -85,B 0,C 180,E1 -6340.699,E2 -6340.699} C_VEL
LIN {X 0,Y 495.72,Z 296.232,A -85,B 0,C 180,E1 -6343.695,E2 -6343.695} C_VEL
LIN {X 0,Y 495.726,Z 296.229,A -85,B 0,C 180,E1 -6346.305,E2 -6346.305} C_VEL
LIN {X 0,Y 495.759,Z 296.22,A -85,B 0,C 180,E1 -6349.301,E2 -6349.301} C_VEL
LIN {X 0,Y 495.725,Z 296.24,A -85,B 0,C 180,E1 -6352.439,E2 -6352.439} C_VEL
LIN {X 0,Y 495.779,Z 296.213,A -85,B 0,C 180,E1 -6355.458,E2 -6355.458} C_VEL
LIN {X 0,Y 495.753,Z 296.236,A -85,B 0,C 180,E1 -6358.364,E2 -6358.364} C_VEL
LIN {X 0,Y 495.747,Z 296.225,A -85,B 0,C 180,E1 -6360.77,E2 -6360.77} C_VEL
LIN {X 0,Y 495.092,Z 296.309,A -85,B 0,C 180,E1 -6361.449,E2 -6361.449} C_VEL
LIN {X 0,Y 492.239,Z 296.672,A -85,B 0,C 180,E1 -6362.552,E2 -6362.552} C_VEL
LIN {X 0,Y 489.832,Z 296.969,A -85,B 0,C 180,E1 -6363.44,E2 -6363.44} C_VEL
LIN {X 0,Y 488.815,Z 297.099,A -85,B 0,C 180,E1 -6364.127,E2 -6364.127} C_VEL
LIN {X 0,Y 488.742,Z 297.107,A -85,B 0,C 180,E1 -6364.359,E2 -6364.359} C_VEL
LIN {X 0,Y 488.723,Z 297.106,A -85,B 0,C 180,E1 -6367.154,E2 -6367.154} C_VEL
LIN {X 0,Y 488.721,Z 297.108,A -85,B 0,C 180,E1 -6369.811,E2 -6369.811} C_VEL
LIN {X 0,Y 488.731,Z 297.11,A -85,B 0,C 180,E1 -6372.424,E2 -6372.424} C_VEL
LIN {X 0,Y 488.758,Z 297.102,A -85,B 0,C 180,E1 -6375,E2 -6375} C_VEL
LIN {X 0,Y 488.802,Z 297.1,A -85,B 0,C 180,E1 -6378.388,E2 -6378.388} C_VEL
LIN {X 0,Y 488.814,Z 297.099,A -85,B 0,C 180,E1 -6381.734,E2 -6381.734} C_VEL
LIN {X 0,Y 488.853,Z 297.095,A -85,B 0,C 180,E1 -6384.224,E2 -6384.224} C_VEL
LIN {X 0,Y 488.959,Z 297.079,A -85,B 0,C 180,E1 -6387.529,E2 -6387.529} C_VEL
LIN {X 0,Y 488.951,Z 297.078,A -85,B 0,C 180,E1 -6390.824,E2 -6390.824} C_VEL
LIN {X 0,Y 488.959,Z 297.079,A -85,B 0,C 180,E1 -6392.471,E2 -6392.471} C_VEL
LIN {X 0,Y 488.852,Z 297.095,A -85,B 0,C 180,E1 -6395.776,E2 -6395.776} C_VEL
LIN {X 0,Y 488.814,Z 297.099,A -85,B 0,C 180,E1 -6398.266,E2 -6398.266} C_VEL
LIN {X 0,Y 488.802,Z 297.1,A -85,B 0,C 180,E1 -6401.612,E2 -6401.612} C_VEL
LIN {X 0,Y 488.758,Z 297.102,A -85,B 0,C 180,E1 -6405,E2 -6405} C_VEL
LIN {X 0,Y 488.75,Z 297.103,A -85,B 0,C 180,E1 -6408.442,E2 -6408.442} C_VEL
LIN {X 0,Y 488.702,Z 297.109,A -85,B 0,C 180,E1 -6411.07,E2 -6411.07} C_VEL
LIN {X 0,Y 488.689,Z 297.116,A -85,B 0,C 180,E1 -6413.745,E2 -6413.745} C_VEL
LIN {X 0,Y 488.793,Z 297.097,A -85,B 0,C 180,E1 -6416.945,E2 -6416.945} C_VEL
LIN {X 0,Y 488.704,Z 297.105,A -85,B 0,C 180,E1 -6420.363,E2 -6420.363} C_VEL
LIN {X 0,Y 488.73,Z 297.1,A -85,B 0,C 180,E1 -6423.484,E2 -6423.484} C_VEL
LIN {X 0,Y 488.682,Z 297.107,A -85,B 0,C 180,E1 -6426.355,E2 -6426.355} C_VEL
LIN {X 0,Y 488.722,Z 297.109,A -85,B 0,C 180,E1 -6429.251,E2 -6429.251} C_VEL
LIN {X 0,Y 488.687,Z 297.09,A -85,B 0,C 180,E1 -6432.525,E2 -6432.525} C_VEL
LIN {X 0,Y 488.703,Z 297.107,A -85,B 0,C 180,E1 -6435.198,E2 -6435.198} C_VEL
LIN {X 0,Y 488.717,Z 297.101,A -85,B 0,C 180,E1 -6438.397,E2 -6438.397} C_VEL
LIN {X 0,Y 488.732,Z 297.103,A -85,B 0,C 180,E1 -6440.942,E2 -6440.942} C_VEL
LIN {X 0,Y 488.676,Z 297.107,A -85,B 0,C 180,E1 -6443.868,E2 -6443.868} C_VEL
LIN {X 0,Y 488.73,Z 297.101,A -85,B 0,C 180,E1 -6446.877,E2 -6446.877} C_VEL
LIN {X 0,Y 488.724,Z 297.104,A -85,B 0,C 180,E1 -6449.781,E2 -6449.781} C_VEL
LIN {X 0,Y 488.782,Z 297.092,A -85,B 0,C 180,E1 -6453.056,E2 -6453.056} C_VEL
LIN {X 0,Y 488.683,Z 297.108,A -85,B 0,C 180,E1 -6456.255,E2 -6456.255} C_VEL
LIN {X 0,Y 488.735,Z 297.1,A -85,B 0,C 180,E1 -6459.176,E2 -6459.176} C_VEL
LIN {X 0,Y 488.749,Z 297.094,A -85,B 0,C 180,E1 -6461.628,E2 -6461.628} C_VEL
LIN {X 0,Y 488.751,Z 297.108,A -85,B 0,C 180,E1 -6465,E2 -6465} C_VEL
LIN {X 0,Y 488.798,Z 297.091,A -85,B 0,C 180,E1 -6468.388,E2 -6468.388} C_VEL
LIN {X 0,Y 488.807,Z 297.087,A -85,B 0,C 180,E1 -6471.734,E2 -6471.734} C_VEL
LIN {X 0,Y 488.845,Z 297.089,A -85,B 0,C 180,E1 -6474.225,E2 -6474.225} C_VEL
LIN {X 0,Y 488.951,Z 297.069,A -85,B 0,C 180,E1 -6477.529,E2 -6477.529} C_VEL
LIN {X 0,Y 488.946,Z 297.07,A -85,B 0,C 180,E1 -6480.824,E2 -6480.824} C_VEL
LIN {X 0,Y 488.951,Z 297.074,A -85,B 0,C 180,E1 -6482.472,E2 -6482.472} C_VEL
LIN {X 0,Y 488.846,Z 297.087,A -85,B 0,C 180,E1 -6485.776,E2 -6485.776} C_VEL
LIN {X 0,Y 488.809,Z 297.089,A -85,B 0,C 180,E1 -6488.267,E2 -6488.267} C_VEL
LIN {X 0,Y 488.799,Z 297.088,A -85,B 0,C 180,E1 -6491.613,E2 -6491.613} C_VEL
LIN {X 0,Y 488.756,Z 297.099,A -85,B 0,C 180,E1 -6495.001,E2 -6495.001} C_VEL
LIN {X 0,Y 488.747,Z 297.094,A -85,B 0,C 180,E1 -6498.443,E2 -6498.443} C_VEL
LIN {X 0,Y 488.699,Z 297.106,A -85,B 0,C 180,E1 -6501.072,E2 -6501.072} C_VEL
LIN {X 0,Y 488.668,Z 297.11,A -85,B 0,C 180,E1 -6503.747,E2 -6503.747} C_VEL
LIN {X 0,Y 488.785,Z 297.089,A -85,B 0,C 180,E1 -6506.945,E2 -6506.945} C_VEL
LIN {X 0,Y 488.703,Z 297.114,A -85,B 0,C 180,E1 -6510.364,E2 -6510.364} C_VEL
LIN {X 0,Y 488.704,Z 297.1,A -85,B 0,C 180,E1 -6513.481,E2 -6513.481} C_VEL
LIN {X 0,Y 488.676,Z 297.116,A -85,B 0,C 180,E1 -6516.355,E2 -6516.355} C_VEL
LIN {X 0,Y 488.695,Z 297.103,A -85,B 0,C 180,E1 -6519.255,E2 -6519.255} C_VEL
LIN {X 0,Y 488.703,Z 297.106,A -85,B 0,C 180,E1 -6521.601,E2 -6521.601} C_VEL
LIN {X 0,Y 488.697,Z 297.107,A -85,B 0,C 180,E1 -6524.804,E2 -6524.804} C_VEL
LIN {X 0,Y 488.688,Z 297.109,A -85,B 0,C 180,E1 -6527.475,E2 -6527.475} C_VEL
LIN {X 0,Y 488.698,Z 297.107,A -85,B 0,C 180,E1 -6530.747,E2 -6530.747} C_VEL
LIN {X 0,Y 488.668,Z 297.111,A -85,B 0,C 180,E1 -6533.868,E2 -6533.868} C_VEL
LIN {X 0,Y 488.737,Z 297.101,A -85,B 0,C 180,E1 -6536.878,E2 -6536.878} C_VEL
LIN {X 0,Y 488.724,Z 297.108,A -85,B 0,C 180,E1 -6539.782,E2 -6539.782} C_VEL
LIN {X 0,Y 488.808,Z 297.194,A -85,B 0,C 180,E1 -6543.054,E2 -6543.054} C_VEL
LIN {X 0,Y 490.267,Z 305.641,A -85,B 0,C 180,E1 -6545.047,E2 -6545.047} C_VEL
LIN {X 0,Y 490.079,Z 314.178,A -85,B 0,C 180,E1 -6546.908,E2 -6546.908} C_VEL
LIN {X 0,Y 489.614,Z 327.081,A -85,B 0,C 180,E1 -6549.63,E2 -6549.63} C_VEL
LIN {X 0,Y 489.094,Z 342.573,A -85,B 0,C 180,E1 -6552.868,E2 -6552.868} C_VEL
LIN {X 0,Y 488.983,Z 346.688,A -85,B 0,C 180,E1 -6553.714,E2 -6553.714} C_VEL
LIN {X 0,Y 490.588,Z 356.205,A -85,B 0,C 180,E1 -6553.94,E2 -6553.94} C_VEL
LIN {X 0,Y 491.705,Z 364.231,A -85,B 0,C 180,E1 -6554.096,E2 -6554.096} C_VEL
LIN {X 0,Y 491.148,Z 451.519,A -85,B 0,C 180,E1 -6555.393,E2 -6555.393} C_VEL
LIN {X 0,Y 490.916,Z 462.285,A -85,B 0,C 180,E1 -6555.65,E2 -6555.65} C_VEL
LIN {X 0,Y 490.708,Z 471.387,A -85,B 0,C 180,E1 -6555.961,E2 -6555.961} C_VEL
LIN {X 0,Y 490.323,Z 481.749,A -85,B 0,C 180,E1 -6556.426,E2 -6556.426} C_VEL
LIN {X 0,Y 490.033,Z 491.183,A -85,B 0,C 180,E1 -6556.965,E2 -6556.965} C_VEL
LIN {X 0,Y 489.698,Z 499.884,A -85,B 0,C 180,E1 -6557.569,E2 -6557.569} C_VEL
LIN {X 0,Y 489.411,Z 508.616,A -85,B 0,C 180,E1 -6558.297,E2 -6558.297} C_VEL
LIN {X 0,Y 489.118,Z 516.012,A -85,B 0,C 180,E1 -6559.025,E2 -6559.025} C_VEL
LIN {X 0,Y 488.8,Z 523.232,A -85,B 0,C 180,E1 -6559.856,E2 -6559.856} C_VEL
LIN {X 0,Y 488.571,Z 529.435,A -85,B 0,C 180,E1 -6560.687,E2 -6560.687} C_VEL
LIN {X 0,Y 488.33,Z 535.972,A -85,B 0,C 180,E1 -6561.726,E2 -6561.726} C_VEL
LIN {X 0,Y 488.2,Z 540.473,A -85,B 0,C 180,E1 -6562.556,E2 -6562.556} C_VEL
LIN {X 0,Y 488.021,Z 545.946,A -85,B 0,C 180,E1 -6563.796,E2 -6563.796} C_VEL
LIN {X 0,Y 487.97,Z 550.283,A -85,B 0,C 180,E1 -6565.043,E2 -6565.043} C_VEL
LIN {X 0,Y 487.929,Z 552.647,A -85,B 0,C 180,E1 -6565.87,E2 -6565.87} C_VEL
LIN {X 0,Y 487.965,Z 554.444,A -85,B 0,C 180,E1 -6566.697,E2 -6566.697} C_VEL
LIN {X 0,Y 487.891,Z 556.883,A -85,B 0,C 180,E1 -6568.349,E2 -6568.349} C_VEL
LIN {X 0,Y 487.834,Z 557.468,A -85,B 0,C 180,E1 -6569.175,E2 -6569.175} C_VEL
LIN {X 0,Y 487.834,Z 557.468,A -85,B 0,C 180,E1 -6570.825,E2 -6570.825} C_VEL
LIN {X 0,Y 487.891,Z 556.883,A -85,B 0,C 180,E1 -6571.651,E2 -6571.651} C_VEL
LIN {X 0,Y 487.965,Z 554.444,A -85,B 0,C 180,E1 -6573.303,E2 -6573.303} C_VEL
LIN {X 0,Y 487.924,Z 551.498,A -85,B 0,C 180,E1 -6574.544,E2 -6574.544} C_VEL
LIN {X 0,Y 488.017,Z 547.515,A -85,B 0,C 180,E1 -6575.786,E2 -6575.786} C_VEL
LIN {X 0,Y 488.098,Z 544.303,A -85,B 0,C 180,E1 -6576.614,E2 -6576.614} C_VEL
LIN {X 0,Y 488.244,Z 538.283,A -85,B 0,C 180,E1 -6577.859,E2 -6577.859} C_VEL
LIN {X 0,Y 488.455,Z 532.187,A -85,B 0,C 180,E1 -6578.898,E2 -6578.898} C_VEL
LIN {X 0,Y 488.685,Z 526.487,A -85,B 0,C 180,E1 -6579.728,E2 -6579.728} C_VEL
LIN {X 0,Y 488.997,Z 517.931,A -85,B 0,C 180,E1 -6580.768,E2 -6580.768} C_VEL
LIN {X 0,Y 489.361,Z 509.751,A -85,B 0,C 180,E1 -6581.599,E2 -6581.599} C_VEL
LIN {X 0,Y 489.621,Z 501.235,A -85,B 0,C 180,E1 -6582.328,E2 -6582.328} C_VEL
LIN {X 0,Y 489.954,Z 492.927,A -85,B 0,C 180,E1 -6582.925,E2 -6582.925} C_VEL
LIN {X 0,Y 490.296,Z 482.756,A -85,B 0,C 180,E1 -6583.522,E2 -6583.522} C_VEL
LIN {X 0,Y 490.647,Z 472.674,A -85,B 0,C 180,E1 -6583.988,E2 -6583.988} C_VEL
LIN {X 0,Y 490.899,Z 463.16,A -85,B 0,C 180,E1 -6584.324,E2 -6584.324} C_VEL
LIN {X 0,Y 491.134,Z 452.851,A -85,B 0,C 180,E1 -6584.581,E2 -6584.581} C_VEL
LIN {X 0,Y 491.567,Z 383.613,A -85,B 0,C 180,E1 -6585.62,E2 -6585.62} C_VEL
LIN {X 0,Y 491.553,Z 362.256,A -85,B 0,C 180,E1 -6585.938,E2 -6585.938} C_VEL
LIN {X 0,Y 489.024,Z 346.819,A -85,B 0,C 180,E1 -6586.275,E2 -6586.275} C_VEL
LIN {X 0,Y 489,Z 346.003,A -85,B 0,C 180,E1 -6586.383,E2 -6586.383} C_VEL
LIN {X 0,Y 489.437,Z 332.387,A -85,B 0,C 180,E1 -6589.284,E2 -6589.284} C_VEL
LIN {X 0,Y 489.928,Z 318.789,A -85,B 0,C 180,E1 -6592.12,E2 -6592.12} C_VEL
LIN {X 0,Y 490.354,Z 307.428,A -85,B 0,C 180,E1 -6594.559,E2 -6594.559} C_VEL
LIN {X 0,Y 489.544,Z 301.261,A -85,B 0,C 180,E1 -6595.967,E2 -6595.967} C_VEL
LIN {X 0,Y 488.804,Z 297.126,A -85,B 0,C 180,E1 -6596.975,E2 -6596.975} C_VEL
LIN {X 0,Y 488.709,Z 297.11,A -85,B 0,C 180,E1 -6600.362,E2 -6600.362} C_VEL
LIN {X 0,Y 488.734,Z 297.103,A -85,B 0,C 180,E1 -6603.483,E2 -6603.483} C_VEL
LIN {X 0,Y 488.671,Z 297.112,A -85,B 0,C 180,E1 -6606.352,E2 -6606.352} C_VEL
LIN {X 0,Y 488.698,Z 297.107,A -85,B 0,C 180,E1 -6609.253,E2 -6609.253} C_VEL
LIN {X 0,Y 488.688,Z 297.109,A -85,B 0,C 180,E1 -6612.525,E2 -6612.525} C_VEL
LIN {X 0,Y 488.697,Z 297.107,A -85,B 0,C 180,E1 -6615.196,E2 -6615.196} C_VEL
LIN {X 0,Y 488.704,Z 297.105,A -85,B 0,C 180,E1 -6618.584,E2 -6618.584} C_VEL
LIN {X 0,Y 488.699,Z 297.103,A -85,B 0,C 180,E1 -6620.946,E2 -6620.946} C_VEL
LIN {X 0,Y 488.672,Z 297.113,A -85,B 0,C 180,E1 -6623.867,E2 -6623.867} C_VEL
LIN {X 0,Y 488.696,Z 297.101,A -85,B 0,C 180,E1 -6626.873,E2 -6626.873} C_VEL
LIN {X 0,Y 488.717,Z 297.109,A -85,B 0,C 180,E1 -6629.78,E2 -6629.78} C_VEL
LIN {X 0,Y 488.785,Z 297.089,A -85,B 0,C 180,E1 -6633.055,E2 -6633.055} C_VEL
LIN {X 0,Y 488.668,Z 297.11,A -85,B 0,C 180,E1 -6636.253,E2 -6636.253} C_VEL
LIN {X 0,Y 488.738,Z 297.103,A -85,B 0,C 180,E1 -6639.175,E2 -6639.175} C_VEL
LIN {X 0,Y 488.751,Z 297.094,A -85,B 0,C 180,E1 -6641.627,E2 -6641.627} C_VEL
LIN {X 0,Y 488.756,Z 297.099,A -85,B 0,C 180,E1 -6644.999,E2 -6644.999} C_VEL
LIN {X 0,Y 488.799,Z 297.088,A -85,B 0,C 180,E1 -6648.387,E2 -6648.387} C_VEL
LIN {X 0,Y 488.809,Z 297.089,A -85,B 0,C 180,E1 -6651.733,E2 -6651.733} C_VEL
LIN {X 0,Y 488.846,Z 297.087,A -85,B 0,C 180,E1 -6654.224,E2 -6654.224} C_VEL
LIN {X 0,Y 488.951,Z 297.074,A -85,B 0,C 180,E1 -6657.528,E2 -6657.528} C_VEL
LIN {X 0,Y 488.957,Z 297.059,A -85,B 0,C 180,E1 -6660,E2 -6660} C_VEL
LIN {X 0,Y 488.951,Z 297.069,A -85,B 0,C 180,E1 -6662.471,E2 -6662.471} C_VEL
LIN {X 0,Y 488.845,Z 297.089,A -85,B 0,C 180,E1 -6665.775,E2 -6665.775} C_VEL
LIN {X 0,Y 488.807,Z 297.087,A -85,B 0,C 180,E1 -6668.266,E2 -6668.266} C_VEL
LIN {X 0,Y 488.798,Z 297.091,A -85,B 0,C 180,E1 -6671.612,E2 -6671.612} C_VEL
LIN {X 0,Y 488.751,Z 297.108,A -85,B 0,C 180,E1 -6675,E2 -6675} C_VEL
LIN {X 0,Y 488.744,Z 297.095,A -85,B 0,C 180,E1 -6678.442,E2 -6678.442} C_VEL
LIN {X 0,Y 488.696,Z 297.109,A -85,B 0,C 180,E1 -6681.071,E2 -6681.071} C_VEL
LIN {X 0,Y 488.682,Z 297.108,A -85,B 0,C 180,E1 -6683.745,E2 -6683.745} C_VEL
LIN {X 0,Y 488.782,Z 297.092,A -85,B 0,C 180,E1 -6686.944,E2 -6686.944} C_VEL
LIN {X 0,Y 488.724,Z 297.104,A -85,B 0,C 180,E1 -6690.219,E2 -6690.219} C_VEL
LIN {X 0,Y 488.726,Z 297.098,A -85,B 0,C 180,E1 -6693.485,E2 -6693.485} C_VEL
LIN {X 0,Y 488.679,Z 297.109,A -85,B 0,C 180,E1 -6696.356,E2 -6696.356} C_VEL
LIN {X 0,Y 488.733,Z 297.101,A -85,B 0,C 180,E1 -6699.25,E2 -6699.25} C_VEL
LIN {X 0,Y 488.723,Z 297.107,A -85,B 0,C 180,E1 -6702.521,E2 -6702.521} C_VEL
LIN {X 0,Y 488.694,Z 297.103,A -85,B 0,C 180,E1 -6705.976,E2 -6705.976} C_VEL
LIN {X 0,Y 488.71,Z 297.092,A -85,B 0,C 180,E1 -6708.586,E2 -6708.586} C_VEL
LIN {X 0,Y 488.697,Z 297.11,A -85,B 0,C 180,E1 -6710.948,E2 -6710.948} C_VEL
LIN {X 0,Y 488.678,Z 297.108,A -85,B 0,C 180,E1 -6713.869,E2 -6713.869} C_VEL
LIN {X 0,Y 488.733,Z 297.105,A -85,B 0,C 180,E1 -6716.878,E2 -6716.878} C_VEL
LIN {X 0,Y 488.718,Z 297.104,A -85,B 0,C 180,E1 -6719.781,E2 -6719.781} C_VEL
LIN {X 0,Y 488.793,Z 297.097,A -85,B 0,C 180,E1 -6723.055,E2 -6723.055} C_VEL
LIN {X 0,Y 488.742,Z 297.107,A -85,B 0,C 180,E1 -6724.359,E2 -6724.359} C_VEL
LIN {X 0,Y 488.095,Z 297.194,A -85,B 0,C 180,E1 -6725.047,E2 -6725.047} C_VEL
LIN {X 0,Y 485.226,Z 297.551,A -85,B 0,C 180,E1 -6726.163,E2 -6726.163} C_VEL
LIN {X 0,Y 482.78,Z 297.85,A -85,B 0,C 180,E1 -6727.063,E2 -6727.063} C_VEL
LIN {X 0,Y 481.722,Z 297.98,A -85,B 0,C 180,E1 -6727.758,E2 -6727.758} C_VEL
LIN {X 0,Y 481.633,Z 297.989,A -85,B 0,C 180,E1 -6727.994,E2 -6727.994} C_VEL
LIN {X 0,Y 481.701,Z 297.985,A -85,B 0,C 180,E1 -6730.393,E2 -6730.393} C_VEL
LIN {X 0,Y 481.688,Z 297.983,A -85,B 0,C 180,E1 -6733.034,E2 -6733.034} C_VEL
LIN {X 0,Y 481.686,Z 297.985,A -85,B 0,C 180,E1 -6735.639,E2 -6735.639} C_VEL
LIN {X 0,Y 481.747,Z 297.98,A -85,B 0,C 180,E1 -6738.215,E2 -6738.215} C_VEL
LIN {X 0,Y 481.759,Z 297.976,A -85,B 0,C 180,E1 -6741.612,E2 -6741.612} C_VEL
LIN {X 0,Y 481.814,Z 297.971,A -85,B 0,C 180,E1 -6744.14,E2 -6744.14} C_VEL
LIN {X 0,Y 481.926,Z 297.955,A -85,B 0,C 180,E1 -6747.493,E2 -6747.493} C_VEL
LIN {X 0,Y 481.902,Z 297.957,A -85,B 0,C 180,E1 -6750.836,E2 -6750.836} C_VEL
LIN {X 0,Y 481.925,Z 297.955,A -85,B 0,C 180,E1 -6752.507,E2 -6752.507} C_VEL
LIN {X 0,Y 481.814,Z 297.971,A -85,B 0,C 180,E1 -6755.86,E2 -6755.86} C_VEL
LIN {X 0,Y 481.759,Z 297.976,A -85,B 0,C 180,E1 -6758.388,E2 -6758.388} C_VEL
LIN {X 0,Y 481.747,Z 297.98,A -85,B 0,C 180,E1 -6761.785,E2 -6761.785} C_VEL
LIN {X 0,Y 481.738,Z 297.978,A -85,B 0,C 180,E1 -6765.224,E2 -6765.224} C_VEL
LIN {X 0,Y 481.708,Z 297.98,A -85,B 0,C 180,E1 -6768.721,E2 -6768.721} C_VEL
LIN {X 0,Y 481.642,Z 297.992,A -85,B 0,C 180,E1 -6771.394,E2 -6771.394} C_VEL
LIN {X 0,Y 481.673,Z 297.986,A -85,B 0,C 180,E1 -6774.113,E2 -6774.113} C_VEL
LIN {X 0,Y 481.746,Z 297.976,A -85,B 0,C 180,E1 -6777.14,E2 -6777.14} C_VEL
LIN {X 0,Y 481.673,Z 297.98,A -85,B 0,C 180,E1 -6779.741,E2 -6779.741} C_VEL
LIN {X 0,Y 481.667,Z 297.983,A -85,B 0,C 180,E1 -6782.674,E2 -6782.674} C_VEL
LIN {X 0,Y 481.636,Z 297.984,A -85,B 0,C 180,E1 -6785.709,E2 -6785.709} C_VEL
LIN {X 0,Y 481.664,Z 297.985,A -85,B 0,C 180,E1 -6788.859,E2 -6788.859} C_VEL
LIN {X 0,Y 481.654,Z 297.966,A -85,B 0,C 180,E1 -6791.914,E2 -6791.914} C_VEL
LIN {X 0,Y 481.652,Z 297.979,A -85,B 0,C 180,E1 -6794.457,E2 -6794.457} C_VEL
LIN {X 0,Y 481.664,Z 297.982,A -85,B 0,C 180,E1 -6797.842,E2 -6797.842} C_VEL
LIN {X 0,Y 481.688,Z 297.983,A -85,B 0,C 180,E1 -6801.143,E2 -6801.143} C_VEL
LIN {X 0,Y 481.659,Z 297.983,A -85,B 0,C 180,E1 -6804.794,E2 -6804.794} C_VEL
LIN {X 0,Y 481.663,Z 297.988,A -85,B 0,C 180,E1 -6807.326,E2 -6807.326} C_VEL
LIN {X 0,Y 481.678,Z 297.98,A -85,B 0,C 180,E1 -6810.259,E2 -6810.259} C_VEL
LIN {X 0,Y 481.735,Z 297.97,A -85,B 0,C 180,E1 -6813.112,E2 -6813.112} C_VEL
LIN {X 0,Y 481.666,Z 297.983,A -85,B 0,C 180,E1 -6815.887,E2 -6815.887} C_VEL
LIN {X 0,Y 481.692,Z 297.979,A -85,B 0,C 180,E1 -6819.028,E2 -6819.028} C_VEL
LIN {X 0,Y 481.697,Z 297.971,A -85,B 0,C 180,E1 -6822.159,E2 -6822.159} C_VEL
LIN {X 0,Y 481.732,Z 297.979,A -85,B 0,C 180,E1 -6824.776,E2 -6824.776} C_VEL
LIN {X 0,Y 481.742,Z 297.968,A -85,B 0,C 180,E1 -6828.215,E2 -6828.215} C_VEL
LIN {X 0,Y 481.753,Z 297.966,A -85,B 0,C 180,E1 -6831.612,E2 -6831.612} C_VEL
LIN {X 0,Y 481.806,Z 297.965,A -85,B 0,C 180,E1 -6834.14,E2 -6834.14} C_VEL
LIN {X 0,Y 481.918,Z 297.945,A -85,B 0,C 180,E1 -6837.493,E2 -6837.493} C_VEL
LIN {X 0,Y 481.897,Z 297.947,A -85,B 0,C 180,E1 -6840.836,E2 -6840.836} C_VEL
LIN {X 0,Y 481.918,Z 297.951,A -85,B 0,C 180,E1 -6842.508,E2 -6842.508} C_VEL
LIN {X 0,Y 481.807,Z 297.964,A -85,B 0,C 180,E1 -6845.861,E2 -6845.861} C_VEL
LIN {X 0,Y 481.755,Z 297.968,A -85,B 0,C 180,E1 -6848.389,E2 -6848.389} C_VEL
LIN {X 0,Y 481.743,Z 297.967,A -85,B 0,C 180,E1 -6851.786,E2 -6851.786} C_VEL
LIN {X 0,Y 481.735,Z 297.972,A -85,B 0,C 180,E1 -6855.225,E2 -6855.225} C_VEL
LIN {X 0,Y 481.704,Z 297.97,A -85,B 0,C 180,E1 -6858.722,E2 -6858.722} C_VEL
LIN {X 0,Y 481.637,Z 297.984,A -85,B 0,C 180,E1 -6861.396,E2 -6861.396} C_VEL
LIN {X 0,Y 481.65,Z 297.987,A -85,B 0,C 180,E1 -6864.115,E2 -6864.115} C_VEL
LIN {X 0,Y 481.74,Z 297.965,A -85,B 0,C 180,E1 -6867.14,E2 -6867.14} C_VEL
LIN {X 0,Y 481.672,Z 297.982,A -85,B 0,C 180,E1 -6869.742,E2 -6869.742} C_VEL
LIN {X 0,Y 481.646,Z 297.982,A -85,B 0,C 180,E1 -6872.677,E2 -6872.677} C_VEL
LIN {X 0,Y 481.63,Z 297.985,A -85,B 0,C 180,E1 -6875.711,E2 -6875.711} C_VEL
LIN {X 0,Y 481.665,Z 297.98,A -85,B 0,C 180,E1 -6878.86,E2 -6878.86} C_VEL
LIN {X 0,Y 481.648,Z 297.988,A -85,B 0,C 180,E1 -6881.914,E2 -6881.914} C_VEL
LIN {X 0,Y 481.651,Z 297.987,A -85,B 0,C 180,E1 -6884.459,E2 -6884.459} C_VEL
LIN {X 0,Y 481.642,Z 297.99,A -85,B 0,C 180,E1 -6887.84,E2 -6887.84} C_VEL
LIN {X 0,Y 481.657,Z 297.985,A -85,B 0,C 180,E1 -6890.655,E2 -6890.655} C_VEL
LIN {X 0,Y 481.62,Z 297.989,A -85,B 0,C 180,E1 -6893.378,E2 -6893.378} C_VEL
LIN {X 0,Y 481.709,Z 297.98,A -85,B 0,C 180,E1 -6896.331,E2 -6896.331} C_VEL
LIN {X 0,Y 481.65,Z 297.99,A -85,B 0,C 180,E1 -6899.418,E2 -6899.418} C_VEL
LIN {X 0,Y 481.711,Z 297.983,A -85,B 0,C 180,E1 -6902.559,E2 -6902.559} C_VEL
LIN {X 0,Y 481.779,Z 298.197,A -85,B 0,C 180,E1 -6902.906,E2 -6902.906} C_VEL
LIN {X 0,Y 483.344,Z 307.289,A -85,B 0,C 180,E1 -6905.061,E2 -6905.061} C_VEL
LIN {X 0,Y 483.017,Z 317.597,A -85,B 0,C 180,E1 -6907.321,E2 -6907.321} C_VEL
LIN {X 0,Y 482.453,Z 331.046,A -85,B 0,C 180,E1 -6910.204,E2 -6910.204} C_VEL
LIN {X 0,Y 482.028,Z 344.362,A -85,B 0,C 180,E1 -6913.047,E2 -6913.047} C_VEL
LIN {X 0,Y 481.985,Z 346.501,A -85,B 0,C 180,E1 -6913.471,E2 -6913.471} C_VEL
LIN {X 0,Y 483.642,Z 356.311,A -85,B 0,C 180,E1 -6913.708,E2 -6913.708} C_VEL
LIN {X 0,Y 484.879,Z 364.468,A -85,B 0,C 180,E1 -6913.873,E2 -6913.873} C_VEL
LIN {X 0,Y 484.283,Z 451.325,A -85,B 0,C 180,E1 -6915.181,E2 -6915.181} C_VEL
LIN {X 0,Y 484.017,Z 462.091,A -85,B 0,C 180,E1 -6915.441,E2 -6915.441} C_VEL
LIN {X 0,Y 483.821,Z 471.193,A -85,B 0,C 180,E1 -6915.757,E2 -6915.757} C_VEL
LIN {X 0,Y 483.426,Z 481.555,A -85,B 0,C 180,E1 -6916.228,E2 -6916.228} C_VEL
LIN {X 0,Y 483.097,Z 490.694,A -85,B 0,C 180,E1 -6916.755,E2 -6916.755} C_VEL
LIN {X 0,Y 482.723,Z 499.689,A -85,B 0,C 180,E1 -6917.386,E2 -6917.386} C_VEL
LIN {X 0,Y 482.436,Z 508.421,A -85,B 0,C 180,E1 -6918.126,E2 -6918.126} C_VEL
LIN {X 0,Y 482.124,Z 515.818,A -85,B 0,C 180,E1 -6918.864,E2 -6918.864} C_VEL
LIN {X 0,Y 481.758,Z 523.037,A -85,B 0,C 180,E1 -6919.706,E2 -6919.706} C_VEL
LIN {X 0,Y 481.515,Z 529.24,A -85,B 0,C 180,E1 -6920.549,E2 -6920.549} C_VEL
LIN {X 0,Y 481.274,Z 535.777,A -85,B 0,C 180,E1 -6921.603,E2 -6921.603} C_VEL
LIN {X 0,Y 481.116,Z 540.278,A -85,B 0,C 180,E1 -6922.446,E2 -6922.446} C_VEL
LIN {X 0,Y 480.922,Z 546.213,A -85,B 0,C 180,E1 -6923.829,E2 -6923.829} C_VEL
LIN {X 0,Y 480.9,Z 550.089,A -85,B 0,C 180,E1 -6924.97,E2 -6924.97} C_VEL
LIN {X 0,Y 480.829,Z 552.452,A -85,B 0,C 180,E1 -6925.809,E2 -6925.809} C_VEL
LIN {X 0,Y 480.889,Z 554.25,A -85,B 0,C 180,E1 -6926.649,E2 -6926.649} C_VEL
LIN {X 0,Y 480.793,Z 556.689,A -85,B 0,C 180,E1 -6928.325,E2 -6928.325} C_VEL
LIN {X 0,Y 480.76,Z 557.275,A -85,B 0,C 180,E1 -6929.162,E2 -6929.162} C_VEL
LIN {X 0,Y 480.76,Z 557.275,A -85,B 0,C 180,E1 -6930.838,E2 -6930.838} C_VEL
LIN {X 0,Y 480.793,Z 556.689,A -85,B 0,C 180,E1 -6931.675,E2 -6931.675} C_VEL
LIN {X 0,Y 480.889,Z 554.25,A -85,B 0,C 180,E1 -6933.351,E2 -6933.351} C_VEL
LIN {X 0,Y 480.842,Z 551.304,A -85,B 0,C 180,E1 -6934.611,E2 -6934.611} C_VEL
LIN {X 0,Y 480.921,Z 547.32,A -85,B 0,C 180,E1 -6935.871,E2 -6935.871} C_VEL
LIN {X 0,Y 481.014,Z 544.108,A -85,B 0,C 180,E1 -6936.712,E2 -6936.712} C_VEL
LIN {X 0,Y 481.197,Z 538.088,A -85,B 0,C 180,E1 -6937.975,E2 -6937.975} C_VEL
LIN {X 0,Y 481.409,Z 531.992,A -85,B 0,C 180,E1 -6939.029,E2 -6939.029} C_VEL
LIN {X 0,Y 481.657,Z 526.292,A -85,B 0,C 180,E1 -6939.872,E2 -6939.872} C_VEL
LIN {X 0,Y 482.002,Z 517.736,A -85,B 0,C 180,E1 -6940.926,E2 -6940.926} C_VEL
LIN {X 0,Y 482.373,Z 509.556,A -85,B 0,C 180,E1 -6941.769,E2 -6941.769} C_VEL
LIN {X 0,Y 482.63,Z 502.393,A -85,B 0,C 180,E1 -6942.403,E2 -6942.403} C_VEL
LIN {X 0,Y 483.042,Z 492.328,A -85,B 0,C 180,E1 -6943.14,E2 -6943.14} C_VEL
LIN {X 0,Y 483.395,Z 482.562,A -85,B 0,C 180,E1 -6943.719,E2 -6943.719} C_VEL
LIN {X 0,Y 483.757,Z 472.48,A -85,B 0,C 180,E1 -6944.191,E2 -6944.191} C_VEL
LIN {X 0,Y 484.027,Z 462.966,A -85,B 0,C 180,E1 -6944.532,E2 -6944.532} C_VEL
LIN {X 0,Y 484.268,Z 452.657,A -85,B 0,C 180,E1 -6944.793,E2 -6944.793} C_VEL
LIN {X 0,Y 484.742,Z 383.21,A -85,B 0,C 180,E1 -6945.849,E2 -6945.849} C_VEL
LIN {X 0,Y 484.694,Z 362.922,A -85,B 0,C 180,E1 -6946.157,E2 -6946.157} C_VEL
LIN {X 0,Y 482.015,Z 346.586,A -85,B 0,C 180,E1 -6946.522,E2 -6946.522} C_VEL
LIN {X 0,Y 482.017,Z 344.361,A -85,B 0,C 180,E1 -6946.954,E2 -6946.954} C_VEL
LIN {X 0,Y 482.545,Z 330.163,A -85,B 0,C 180,E1 -6950.014,E2 -6950.014} C_VEL
LIN {X 0,Y 483.002,Z 317.606,A -85,B 0,C 180,E1 -6952.68,E2 -6952.68} C_VEL
LIN {X 0,Y 483.39,Z 308.312,A -85,B 0,C 180,E1 -6954.707,E2 -6954.707} C_VEL
LIN {X 0,Y 482.118,Z 300.11,A -85,B 0,C 180,E1 -6956.631,E2 -6956.631} C_VEL
LIN {X 0,Y 481.748,Z 297.999,A -85,B 0,C 180,E1 -6957.193,E2 -6957.193} C_VEL
LIN {X 0,Y 481.678,Z 297.984,A -85,B 0,C 180,E1 -6959.74,E2 -6959.74} C_VEL
LIN {X 0,Y 481.671,Z 297.982,A -85,B 0,C 180,E1 -6962.673,E2 -6962.673} C_VEL
LIN {X 0,Y 481.659,Z 297.983,A -85,B 0,C 180,E1 -6965.203,E2 -6965.203} C_VEL
LIN {X 0,Y 481.667,Z 297.982,A -85,B 0,C 180,E1 -6968.858,E2 -6968.858} C_VEL
LIN {X 0,Y 481.644,Z 297.985,A -85,B 0,C 180,E1 -6971.911,E2 -6971.911} C_VEL
LIN {X 0,Y 481.651,Z 297.985,A -85,B 0,C 180,E1 -6974.457,E2 -6974.457} C_VEL
LIN {X 0,Y 481.644,Z 297.992,A -85,B 0,C 180,E1 -6977.838,E2 -6977.838} C_VEL
LIN {X 0,Y 481.656,Z 297.98,A -85,B 0,C 180,E1 -6980.653,E2 -6980.653} C_VEL
LIN {X 0,Y 481.622,Z 297.992,A -85,B 0,C 180,E1 -6983.375,E2 -6983.375} C_VEL
LIN {X 0,Y 481.664,Z 297.978,A -85,B 0,C 180,E1 -6986.326,E2 -6986.326} C_VEL
LIN {X 0,Y 481.644,Z 297.99,A -85,B 0,C 180,E1 -6989.417,E2 -6989.417} C_VEL
LIN {X 0,Y 481.693,Z 297.972,A -85,B 0,C 180,E1 -6992.167,E2 -6992.167} C_VEL
LIN {X 0,Y 481.685,Z 297.976,A -85,B 0,C 180,E1 -6994.968,E2 -6994.968} C_VEL
LIN {X 0,Y 481.641,Z 297.989,A -85,B 0,C 180,E1 -6997.704,E2 -6997.704} C_VEL
LIN {X 0,Y 481.699,Z 297.969,A -85,B 0,C 180,E1 -7000.392,E2 -7000.392} C_VEL
LIN {X 0,Y 481.682,Z 297.974,A -85,B 0,C 180,E1 -7003.033,E2 -7003.033} C_VEL
LIN {X 0,Y 481.686,Z 297.984,A -85,B 0,C 180,E1 -7005.638,E2 -7005.638} C_VEL
LIN {X 0,Y 481.743,Z 297.967,A -85,B 0,C 180,E1 -7008.214,E2 -7008.214} C_VEL
LIN {X 0,Y 481.755,Z 297.968,A -85,B 0,C 180,E1 -7011.611,E2 -7011.611} C_VEL
LIN {X 0,Y 481.807,Z 297.964,A -85,B 0,C 180,E1 -7014.139,E2 -7014.139} C_VEL
LIN {X 0,Y 481.918,Z 297.951,A -85,B 0,C 180,E1 -7017.492,E2 -7017.492} C_VEL
LIN {X 0,Y 481.896,Z 297.941,A -85,B 0,C 180,E1 -7020.835,E2 -7020.835} C_VEL
LIN {X 0,Y 481.918,Z 297.945,A -85,B 0,C 180,E1 -7022.507,E2 -7022.507} C_VEL
LIN {X 0,Y 481.806,Z 297.965,A -85,B 0,C 180,E1 -7025.86,E2 -7025.86} C_VEL
LIN {X 0,Y 481.753,Z 297.966,A -85,B 0,C 180,E1 -7028.388,E2 -7028.388} C_VEL
LIN {X 0,Y 481.742,Z 297.968,A -85,B 0,C 180,E1 -7031.785,E2 -7031.785} C_VEL
LIN {X 0,Y 481.732,Z 297.979,A -85,B 0,C 180,E1 -7035.224,E2 -7035.224} C_VEL
LIN {X 0,Y 481.702,Z 297.973,A -85,B 0,C 180,E1 -7038.722,E2 -7038.722} C_VEL
LIN {X 0,Y 481.635,Z 297.987,A -85,B 0,C 180,E1 -7041.395,E2 -7041.395} C_VEL
LIN {X 0,Y 481.666,Z 297.983,A -85,B 0,C 180,E1 -7044.113,E2 -7044.113} C_VEL
LIN {X 0,Y 481.737,Z 297.968,A -85,B 0,C 180,E1 -7047.139,E2 -7047.139} C_VEL
LIN {X 0,Y 481.678,Z 297.98,A -85,B 0,C 180,E1 -7049.741,E2 -7049.741} C_VEL
LIN {X 0,Y 481.663,Z 297.988,A -85,B 0,C 180,E1 -7052.674,E2 -7052.674} C_VEL
LIN {X 0,Y 481.633,Z 297.983,A -85,B 0,C 180,E1 -7055.709,E2 -7055.709} C_VEL
LIN {X 0,Y 481.705,Z 297.976,A -85,B 0,C 180,E1 -7059.354,E2 -7059.354} C_VEL
LIN {X 0,Y 481.664,Z 297.982,A -85,B 0,C 180,E1 -7062.158,E2 -7062.158} C_VEL
LIN {X 0,Y 481.652,Z 297.979,A -85,B 0,C 180,E1 -7065.543,E2 -7065.543} C_VEL
LIN {X 0,Y 481.654,Z 297.966,A -85,B 0,C 180,E1 -7068.086,E2 -7068.086} C_VEL
LIN {X 0,Y 481.664,Z 297.985,A -85,B 0,C 180,E1 -7071.141,E2 -7071.141} C_VEL
LIN {X 0,Y 481.662,Z 297.973,A -85,B 0,C 180,E1 -7074.795,E2 -7074.795} C_VEL
LIN {X 0,Y 481.667,Z 297.983,A -85,B 0,C 180,E1 -7077.326,E2 -7077.326} C_VEL
LIN {X 0,Y 481.673,Z 297.98,A -85,B 0,C 180,E1 -7080.259,E2 -7080.259} C_VEL
LIN {X 0,Y 481.747,Z 297.975,A -85,B 0,C 180,E1 -7083.113,E2 -7083.113} C_VEL
LIN {X 0,Y 481.673,Z 297.986,A -85,B 0,C 180,E1 -7085.887,E2 -7085.887} C_VEL
LIN {X 0,Y 481.633,Z 297.989,A -85,B 0,C 180,E1 -7087.994,E2 -7087.994} C_VEL
LIN {X 0,Y 480.965,Z 298.076,A -85,B 0,C 180,E1 -7088.692,E2 -7088.692} C_VEL
LIN {X 0,Y 478.136,Z 298.427,A -85,B 0,C 180,E1 -7089.826,E2 -7089.826} C_VEL
LIN {X 0,Y 475.752,Z 298.724,A -85,B 0,C 180,E1 -7090.74,E2 -7090.74} C_VEL
LIN {X 0,Y 474.732,Z 298.849,A -85,B 0,C 180,E1 -7091.446,E2 -7091.446} C_VEL
LIN {X 0,Y 474.651,Z 298.86,A -85,B 0,C 180,E1 -7091.685,E2 -7091.685} C_VEL
LIN {X 0,Y 474.696,Z 298.857,A -85,B 0,C 180,E1 -7094.545,E2 -7094.545} C_VEL
LIN {X 0,Y 474.7,Z 298.857,A -85,B 0,C 180,E1 -7098.038,E2 -7098.038} C_VEL
LIN {X 0,Y 474.724,Z 298.852,A -85,B 0,C 180,E1 -7101.487,E2 -7101.487} C_VEL
LIN {X 0,Y 474.776,Z 298.848,A -85,B 0,C 180,E1 -7104.053,E2 -7104.053} C_VEL
LIN {X 0,Y 474.891,Z 298.831,A -85,B 0,C 180,E1 -7107.455,E2 -7107.455} C_VEL
LIN {X 0,Y 474.909,Z 298.832,A -85,B 0,C 180,E1 -7110,E2 -7110} C_VEL
LIN {X 0,Y 474.891,Z 298.831,A -85,B 0,C 180,E1 -7112.545,E2 -7112.545} C_VEL
LIN {X 0,Y 474.776,Z 298.848,A -85,B 0,C 180,E1 -7115.947,E2 -7115.947} C_VEL
LIN {X 0,Y 474.724,Z 298.852,A -85,B 0,C 180,E1 -7118.513,E2 -7118.513} C_VEL
LIN {X 0,Y 474.7,Z 298.857,A -85,B 0,C 180,E1 -7121.962,E2 -7121.962} C_VEL
LIN {X 0,Y 474.696,Z 298.857,A -85,B 0,C 180,E1 -7125.455,E2 -7125.455} C_VEL
LIN {X 0,Y 474.66,Z 298.858,A -85,B 0,C 180,E1 -7129.01,E2 -7129.01} C_VEL
LIN {X 0,Y 474.586,Z 298.872,A -85,B 0,C 180,E1 -7131.728,E2 -7131.728} C_VEL
LIN {X 0,Y 474.654,Z 298.858,A -85,B 0,C 180,E1 -7134.492,E2 -7134.492} C_VEL
LIN {X 0,Y 474.693,Z 298.857,A -85,B 0,C 180,E1 -7137.338,E2 -7137.338} C_VEL
LIN {X 0,Y 474.599,Z 298.862,A -85,B 0,C 180,E1 -7140.81,E2 -7140.81} C_VEL
LIN {X 0,Y 474.631,Z 298.848,A -85,B 0,C 180,E1 -7143.984,E2 -7143.984} C_VEL
LIN {X 0,Y 474.568,Z 298.866,A -85,B 0,C 180,E1 -7146.9,E2 -7146.9} C_VEL
LIN {X 0,Y 474.636,Z 298.856,A -85,B 0,C 180,E1 -7149.65,E2 -7149.65} C_VEL
LIN {X 0,Y 474.627,Z 298.842,A -85,B 0,C 180,E1 -7152.932,E2 -7152.932} C_VEL
LIN {X 0,Y 474.607,Z 298.864,A -85,B 0,C 180,E1 -7155.896,E2 -7155.896} C_VEL
LIN {X 0,Y 474.636,Z 298.859,A -85,B 0,C 180,E1 -7159.038,E2 -7159.038} C_VEL
LIN {X 0,Y 474.607,Z 298.866,A -85,B 0,C 180,E1 -7161.703,E2 -7161.703} C_VEL
LIN {X 0,Y 474.621,Z 298.859,A -85,B 0,C 180,E1 -7164.726,E2 -7164.726} C_VEL
LIN {X 0,Y 474.628,Z 298.861,A -85,B 0,C 180,E1 -7167.788,E2 -7167.788} C_VEL
LIN {X 0,Y 474.623,Z 298.863,A -85,B 0,C 180,E1 -7170.883,E2 -7170.883} C_VEL
LIN {X 0,Y 474.65,Z 298.854,A -85,B 0,C 180,E1 -7173.628,E2 -7173.628} C_VEL
LIN {X 0,Y 474.625,Z 298.862,A -85,B 0,C 180,E1 -7176.641,E2 -7176.641} C_VEL
LIN {X 0,Y 474.646,Z 298.847,A -85,B 0,C 180,E1 -7180.09,E2 -7180.09} C_VEL
LIN {X 0,Y 474.641,Z 298.854,A -85,B 0,C 180,E1 -7182.775,E2 -7182.775} C_VEL
LIN {X 0,Y 474.638,Z 298.86,A -85,B 0,C 180,E1 -7185.421,E2 -7185.421} C_VEL
LIN {X 0,Y 474.695,Z 298.845,A -85,B 0,C 180,E1 -7188.038,E2 -7188.038} C_VEL
LIN {X 0,Y 474.718,Z 298.843,A -85,B 0,C 180,E1 -7191.487,E2 -7191.487} C_VEL
LIN {X 0,Y 474.769,Z 298.841,A -85,B 0,C 180,E1 -7194.053,E2 -7194.053} C_VEL
LIN {X 0,Y 474.884,Z 298.821,A -85,B 0,C 180,E1 -7197.456,E2 -7197.456} C_VEL
LIN {X 0,Y 474.849,Z 298.825,A -85,B 0,C 180,E1 -7200.849,E2 -7200.849} C_VEL
LIN {X 0,Y 474.884,Z 298.827,A -85,B 0,C 180,E1 -7202.545,E2 -7202.545} C_VEL
LIN {X 0,Y 474.769,Z 298.841,A -85,B 0,C 180,E1 -7205.948,E2 -7205.948} C_VEL
LIN {X 0,Y 474.72,Z 298.841,A -85,B 0,C 180,E1 -7208.514,E2 -7208.514} C_VEL
LIN {X 0,Y 474.696,Z 298.846,A -85,B 0,C 180,E1 -7211.963,E2 -7211.963} C_VEL
LIN {X 0,Y 474.692,Z 298.848,A -85,B 0,C 180,E1 -7215.456,E2 -7215.456} C_VEL
LIN {X 0,Y 474.657,Z 298.847,A -85,B 0,C 180,E1 -7219.011,E2 -7219.011} C_VEL
LIN {X 0,Y 474.58,Z 298.863,A -85,B 0,C 180,E1 -7221.73,E2 -7221.73} C_VEL
LIN {X 0,Y 474.631,Z 298.86,A -85,B 0,C 180,E1 -7224.495,E2 -7224.495} C_VEL
LIN {X 0,Y 474.674,Z 298.844,A -85,B 0,C 180,E1 -7227.335,E2 -7227.335} C_VEL
LIN {X 0,Y 474.599,Z 298.868,A -85,B 0,C 180,E1 -7230.231,E2 -7230.231} C_VEL
LIN {X 0,Y 474.608,Z 298.855,A -85,B 0,C 180,E1 -7233.223,E2 -7233.223} C_VEL
LIN {X 0,Y 474.583,Z 298.871,A -85,B 0,C 180,E1 -7236.325,E2 -7236.325} C_VEL
LIN {X 0,Y 474.613,Z 298.859,A -85,B 0,C 180,E1 -7239.647,E2 -7239.647} C_VEL
LIN {X 0,Y 474.62,Z 298.868,A -85,B 0,C 180,E1 -7242.238,E2 -7242.238} C_VEL
LIN {X 0,Y 474.613,Z 298.86,A -85,B 0,C 180,E1 -7245.299,E2 -7245.299} C_VEL
LIN {X 0,Y 474.613,Z 298.858,A -85,B 0,C 180,E1 -7248.215,E2 -7248.215} C_VEL
LIN {X 0,Y 474.608,Z 298.863,A -85,B 0,C 180,E1 -7251.543,E2 -7251.543} C_VEL
LIN {X 0,Y 474.62,Z 298.86,A -85,B 0,C 180,E1 -7254.726,E2 -7254.726} C_VEL
LIN {X 0,Y 474.635,Z 298.859,A -85,B 0,C 180,E1 -7257.789,E2 -7257.789} C_VEL
LIN {X 0,Y 474.622,Z 298.865,A -85,B 0,C 180,E1 -7260.886,E2 -7260.886} C_VEL
LIN {X 0,Y 474.716,Z 299.018,A -85,B 0,C 180,E1 -7262.682,E2 -7262.682} C_VEL
LIN {X 0,Y 476.344,Z 308.172,A -85,B 0,C 180,E1 -7264.902,E2 -7264.902} C_VEL
LIN {X 0,Y 476.134,Z 316.39,A -85,B 0,C 180,E1 -7266.744,E2 -7266.744} C_VEL
LIN {X 0,Y 475.576,Z 329.845,A -85,B 0,C 180,E1 -7269.679,E2 -7269.679} C_VEL
LIN {X 0,Y 475.008,Z 344.173,A -85,B 0,C 180,E1 -7272.788,E2 -7272.788} C_VEL
LIN {X 0,Y 474.987,Z 346.275,A -85,B 0,C 180,E1 -7273.217,E2 -7273.217} C_VEL
LIN {X 0,Y 476.443,Z 355.039,A -85,B 0,C 180,E1 -7273.438,E2 -7273.438} C_VEL
LIN {X 0,Y 478.06,Z 365.035,A -85,B 0,C 180,E1 -7273.648,E2 -7273.648} C_VEL
LIN {X 0,Y 477.434,Z 451.132,A -85,B 0,C 180,E1 -7274.963,E2 -7274.963} C_VEL
LIN {X 0,Y 477.158,Z 461.897,A -85,B 0,C 180,E1 -7275.227,E2 -7275.227} C_VEL
LIN {X 0,Y 476.945,Z 470.999,A -85,B 0,C 180,E1 -7275.548,E2 -7275.548} C_VEL
LIN {X 0,Y 476.496,Z 481.36,A -85,B 0,C 180,E1 -7276.024,E2 -7276.024} C_VEL
LIN {X 0,Y 476.169,Z 490.499,A -85,B 0,C 180,E1 -7276.559,E2 -7276.559} C_VEL
LIN {X 0,Y 475.765,Z 499.494,A -85,B 0,C 180,E1 -7277.198,E2 -7277.198} C_VEL
LIN {X 0,Y 475.464,Z 508.316,A -85,B 0,C 180,E1 -7277.958,E2 -7277.958} C_VEL
LIN {X 0,Y 475.121,Z 515.623,A -85,B 0,C 180,E1 -7278.697,E2 -7278.697} C_VEL
LIN {X 0,Y 474.746,Z 522.842,A -85,B 0,C 180,E1 -7279.552,E2 -7279.552} C_VEL
LIN {X 0,Y 474.482,Z 529.045,A -85,B 0,C 180,E1 -7280.408,E2 -7280.408} C_VEL
LIN {X 0,Y 474.206,Z 535.582,A -85,B 0,C 180,E1 -7281.477,E2 -7281.477} C_VEL
LIN {X 0,Y 474.043,Z 540.083,A -85,B 0,C 180,E1 -7282.332,E2 -7282.332} C_VEL
LIN {X 0,Y 473.87,Z 545.371,A -85,B 0,C 180,E1 -7283.558,E2 -7283.558} C_VEL
LIN {X 0,Y 473.83,Z 549.896,A -85,B 0,C 180,E1 -7284.894,E2 -7284.894} C_VEL
LIN {X 0,Y 473.736,Z 552.258,A -85,B 0,C 180,E1 -7285.746,E2 -7285.746} C_VEL
LIN {X 0,Y 473.796,Z 554.056,A -85,B 0,C 180,E1 -7286.599,E2 -7286.599} C_VEL
LIN {X 0,Y 473.698,Z 556.495,A -85,B 0,C 180,E1 -7288.3,E2 -7288.3} C_VEL
LIN {X 0,Y 473.688,Z 557.082,A -85,B 0,C 180,E1 -7289.15,E2 -7289.15} C_VEL
LIN {X 0,Y 473.688,Z 557.082,A -85,B 0,C 180,E1 -7290.85,E2 -7290.85} C_VEL
LIN {X 0,Y 473.698,Z 556.495,A -85,B 0,C 180,E1 -7291.7,E2 -7291.7} C_VEL
LIN {X 0,Y 473.796,Z 554.056,A -85,B 0,C 180,E1 -7293.401,E2 -7293.401} C_VEL
LIN {X 0,Y 473.765,Z 551.11,A -85,B 0,C 180,E1 -7294.68,E2 -7294.68} C_VEL
LIN {X 0,Y 473.829,Z 547.125,A -85,B 0,C 180,E1 -7295.959,E2 -7295.959} C_VEL
LIN {X 0,Y 474.005,Z 541.999,A -85,B 0,C 180,E1 -7297.24,E2 -7297.24} C_VEL
LIN {X 0,Y 474.174,Z 536.738,A -85,B 0,C 180,E1 -7298.309,E2 -7298.309} C_VEL
LIN {X 0,Y 474.414,Z 530.421,A -85,B 0,C 180,E1 -7299.378,E2 -7299.378} C_VEL
LIN {X 0,Y 474.65,Z 524.469,A -85,B 0,C 180,E1 -7300.234,E2 -7300.234} C_VEL
LIN {X 0,Y 475.005,Z 517.542,A -85,B 0,C 180,E1 -7301.089,E2 -7301.089} C_VEL
LIN {X 0,Y 475.384,Z 509.361,A -85,B 0,C 180,E1 -7301.945,E2 -7301.945} C_VEL
LIN {X 0,Y 475.684,Z 501.409,A -85,B 0,C 180,E1 -7302.65,E2 -7302.65} C_VEL
LIN {X 0,Y 476.12,Z 492.134,A -85,B 0,C 180,E1 -7303.334,E2 -7303.334} C_VEL
LIN {X 0,Y 476.511,Z 482.369,A -85,B 0,C 180,E1 -7303.921,E2 -7303.921} C_VEL
LIN {X 0,Y 476.84,Z 473.574,A -85,B 0,C 180,E1 -7304.347,E2 -7304.347} C_VEL
LIN {X 0,Y 477.151,Z 463.647,A -85,B 0,C 180,E1 -7304.719,E2 -7304.719} C_VEL
LIN {X 0,Y 477.384,Z 453.795,A -85,B 0,C 180,E1 -7304.984,E2 -7304.984} C_VEL
LIN {X 0,Y 477.64,Z 428.057,A -85,B 0,C 180,E1 -7305.402,E2 -7305.402} C_VEL
LIN {X 0,Y 477.949,Z 364.266,A -85,B 0,C 180,E1 -7306.368,E2 -7306.368} C_VEL
LIN {X 0,Y 474.986,Z 346.47,A -85,B 0,C 180,E1 -7306.768,E2 -7306.768} C_VEL
LIN {X 0,Y 474.958,Z 345.615,A -85,B 0,C 180,E1 -7306.881,E2 -7306.881} C_VEL
LIN {X 0,Y 475.476,Z 333.094,A -85,B 0,C 180,E1 -7309.649,E2 -7309.649} C_VEL
LIN {X 0,Y 475.978,Z 320.612,A -85,B 0,C 180,E1 -7312.346,E2 -7312.346} C_VEL
LIN {X 0,Y 476.418,Z 309.195,A -85,B 0,C 180,E1 -7314.861,E2 -7314.861} C_VEL
LIN {X 0,Y 475.087,Z 300.991,A -85,B 0,C 180,E1 -7316.819,E2 -7316.819} C_VEL
LIN {X 0,Y 474.676,Z 298.883,A -85,B 0,C 180,E1 -7317.398,E2 -7317.398} C_VEL
LIN {X 0,Y 474.604,Z 298.867,A -85,B 0,C 180,E1 -7320.809,E2 -7320.809} C_VEL
LIN {X 0,Y 474.637,Z 298.866,A -85,B 0,C 180,E1 -7323.983,E2 -7323.983} C_VEL
LIN {X 0,Y 474.564,Z 298.867,A -85,B 0,C 180,E1 -7326.897,E2 -7326.897} C_VEL
LIN {X 0,Y 474.605,Z 298.861,A -85,B 0,C 180,E1 -7329.644,E2 -7329.644} C_VEL
LIN {X 0,Y 474.619,Z 298.864,A -85,B 0,C 180,E1 -7332.235,E2 -7332.235} C_VEL
LIN {X 0,Y 474.613,Z 298.862,A -85,B 0,C 180,E1 -7335.297,E2 -7335.297} C_VEL
LIN {X 0,Y 474.617,Z 298.863,A -85,B 0,C 180,E1 -7338.214,E2 -7338.214} C_VEL
LIN {X 0,Y 474.606,Z 298.864,A -85,B 0,C 180,E1 -7341.542,E2 -7341.542} C_VEL
LIN {X 0,Y 474.617,Z 298.857,A -85,B 0,C 180,E1 -7344.725,E2 -7344.725} C_VEL
LIN {X 0,Y 474.621,Z 298.865,A -85,B 0,C 180,E1 -7347.786,E2 -7347.786} C_VEL
LIN {X 0,Y 474.617,Z 298.86,A -85,B 0,C 180,E1 -7350.884,E2 -7350.884} C_VEL
LIN {X 0,Y 474.647,Z 298.852,A -85,B 0,C 180,E1 -7353.627,E2 -7353.627} C_VEL
LIN {X 0,Y 474.627,Z 298.858,A -85,B 0,C 180,E1 -7356.641,E2 -7356.641} C_VEL
LIN {X 0,Y 474.648,Z 298.848,A -85,B 0,C 180,E1 -7360.089,E2 -7360.089} C_VEL
LIN {X 0,Y 474.642,Z 298.848,A -85,B 0,C 180,E1 -7362.774,E2 -7362.774} C_VEL
LIN {X 0,Y 474.644,Z 298.863,A -85,B 0,C 180,E1 -7365.42,E2 -7365.42} C_VEL
LIN {X 0,Y 474.696,Z 298.846,A -85,B 0,C 180,E1 -7368.037,E2 -7368.037} C_VEL
LIN {X 0,Y 474.72,Z 298.841,A -85,B 0,C 180,E1 -7371.486,E2 -7371.486} C_VEL
LIN {X 0,Y 474.769,Z 298.841,A -85,B 0,C 180,E1 -7374.052,E2 -7374.052} C_VEL
LIN {X 0,Y 474.884,Z 298.827,A -85,B 0,C 180,E1 -7377.455,E2 -7377.455} C_VEL
LIN {X 0,Y 474.848,Z 298.818,A -85,B 0,C 180,E1 -7380.848,E2 -7380.848} C_VEL
LIN {X 0,Y 474.884,Z 298.821,A -85,B 0,C 180,E1 -7382.544,E2 -7382.544} C_VEL
LIN {X 0,Y 474.769,Z 298.841,A -85,B 0,C 180,E1 -7385.947,E2 -7385.947} C_VEL
LIN {X 0,Y 474.718,Z 298.843,A -85,B 0,C 180,E1 -7388.513,E2 -7388.513} C_VEL
LIN {X 0,Y 474.695,Z 298.845,A -85,B 0,C 180,E1 -7391.962,E2 -7391.962} C_VEL
LIN {X 0,Y 474.689,Z 298.853,A -85,B 0,C 180,E1 -7395.455,E2 -7395.455} C_VEL
LIN {X 0,Y 474.655,Z 298.848,A -85,B 0,C 180,E1 -7399.01,E2 -7399.01} C_VEL
LIN {X 0,Y 474.578,Z 298.864,A -85,B 0,C 180,E1 -7401.729,E2 -7401.729} C_VEL
LIN {X 0,Y 474.648,Z 298.86,A -85,B 0,C 180,E1 -7404.493,E2 -7404.493} C_VEL
LIN {X 0,Y 474.671,Z 298.847,A -85,B 0,C 180,E1 -7407.334,E2 -7407.334} C_VEL
LIN {X 0,Y 474.604,Z 298.863,A -85,B 0,C 180,E1 -7410.23,E2 -7410.23} C_VEL
LIN {X 0,Y 474.633,Z 298.856,A -85,B 0,C 180,E1 -7413.22,E2 -7413.22} C_VEL
LIN {X 0,Y 474.584,Z 298.864,A -85,B 0,C 180,E1 -7416.323,E2 -7416.323} C_VEL
LIN {X 0,Y 474.641,Z 298.855,A -85,B 0,C 180,E1 -7419.651,E2 -7419.651} C_VEL
LIN {X 0,Y 474.637,Z 298.863,A -85,B 0,C 180,E1 -7422.931,E2 -7422.931} C_VEL
LIN {X 0,Y 474.607,Z 298.857,A -85,B 0,C 180,E1 -7425.896,E2 -7425.896} C_VEL
LIN {X 0,Y 474.624,Z 298.851,A -85,B 0,C 180,E1 -7429.04,E2 -7429.04} C_VEL
LIN {X 0,Y 474.603,Z 298.863,A -85,B 0,C 180,E1 -7431.704,E2 -7431.704} C_VEL
LIN {X 0,Y 474.623,Z 298.85,A -85,B 0,C 180,E1 -7434.727,E2 -7434.727} C_VEL
LIN {X 0,Y 474.631,Z 298.86,A -85,B 0,C 180,E1 -7437.788,E2 -7437.788} C_VEL
LIN {X 0,Y 474.618,Z 298.857,A -85,B 0,C 180,E1 -7440.885,E2 -7440.885} C_VEL
LIN {X 0,Y 474.661,Z 298.858,A -85,B 0,C 180,E1 -7443.629,E2 -7443.629} C_VEL
LIN {X 0,Y 474.631,Z 298.865,A -85,B 0,C 180,E1 -7446.641,E2 -7446.641} C_VEL
LIN {X 0,Y 474.65,Z 298.863,A -85,B 0,C 180,E1 -7450.09,E2 -7450.09} C_VEL
LIN {X 0,Y 474.651,Z 298.86,A -85,B 0,C 180,E1 -7451.685,E2 -7451.685} C_VEL
LIN {X 0,Y 473.989,Z 298.947,A -85,B 0,C 180,E1 -7452.394,E2 -7452.394} C_VEL
LIN {X 0,Y 471.138,Z 299.302,A -85,B 0,C 180,E1 -7453.546,E2 -7453.546} C_VEL
LIN {X 0,Y 468.72,Z 299.602,A -85,B 0,C 180,E1 -7454.474,E2 -7454.474} C_VEL
LIN {X 0,Y 467.679,Z 299.728,A -85,B 0,C 180,E1 -7455.191,E2 -7455.191} C_VEL
LIN {X 0,Y 467.592,Z 299.739,A -85,B 0,C 180,E1 -7455.434,E2 -7455.434} C_VEL
LIN {X 0,Y 467.65,Z 299.734,A -85,B 0,C 180,E1 -7458.734,E2 -7458.734} C_VEL
LIN {X 0,Y 467.745,Z 299.724,A -85,B 0,C 180,E1 -7462.228,E2 -7462.228} C_VEL
LIN {X 0,Y 467.722,Z 299.724,A -85,B 0,C 180,E1 -7464.828,E2 -7464.828} C_VEL
LIN {X 0,Y 467.857,Z 299.708,A -85,B 0,C 180,E1 -7467.417,E2 -7467.417} C_VEL
LIN {X 0,Y 467.88,Z 299.708,A -85,B 0,C 180,E1 -7470,E2 -7470} C_VEL
LIN {X 0,Y 467.857,Z 299.707,A -85,B 0,C 180,E1 -7472.583,E2 -7472.583} C_VEL
LIN {X 0,Y 467.741,Z 299.724,A -85,B 0,C 180,E1 -7476.037,E2 -7476.037} C_VEL
LIN {X 0,Y 467.678,Z 299.729,A -85,B 0,C 180,E1 -7478.643,E2 -7478.643} C_VEL
LIN {X 0,Y 467.652,Z 299.735,A -85,B 0,C 180,E1 -7482.145,E2 -7482.145} C_VEL
LIN {X 0,Y 467.635,Z 299.738,A -85,B 0,C 180,E1 -7485.695,E2 -7485.695} C_VEL
LIN {X 0,Y 467.613,Z 299.736,A -85,B 0,C 180,E1 -7488.764,E2 -7488.764} C_VEL
LIN {X 0,Y 467.576,Z 299.743,A -85,B 0,C 180,E1 -7491.268,E2 -7491.268} C_VEL
LIN {X 0,Y 467.568,Z 299.745,A -85,B 0,C 180,E1 -7493.943,E2 -7493.943} C_VEL
LIN {X 0,Y 467.622,Z 299.734,A -85,B 0,C 180,E1 -7496.799,E2 -7496.799} C_VEL
LIN {X 0,Y 467.548,Z 299.738,A -85,B 0,C 180,E1 -7499.738,E2 -7499.738} C_VEL
LIN {X 0,Y 467.577,Z 299.738,A -85,B 0,C 180,E1 -7502.758,E2 -7502.758} C_VEL
LIN {X 0,Y 467.55,Z 299.74,A -85,B 0,C 180,E1 -7505.889,E2 -7505.889} C_VEL
LIN {X 0,Y 467.585,Z 299.742,A -85,B 0,C 180,E1 -7509.143,E2 -7509.143} C_VEL
LIN {X 0,Y 467.578,Z 299.717,A -85,B 0,C 180,E1 -7512.567,E2 -7512.567} C_VEL
LIN {X 0,Y 467.562,Z 299.738,A -85,B 0,C 180,E1 -7515.053,E2 -7515.053} C_VEL
LIN {X 0,Y 467.585,Z 299.741,A -85,B 0,C 180,E1 -7517.44,E2 -7517.44} C_VEL
LIN {X 0,Y 467.606,Z 299.734,A -85,B 0,C 180,E1 -7520.858,E2 -7520.858} C_VEL
LIN {X 0,Y 467.554,Z 299.737,A -85,B 0,C 180,E1 -7524.26,E2 -7524.26} C_VEL
LIN {X 0,Y 467.573,Z 299.743,A -85,B 0,C 180,E1 -7527.321,E2 -7527.321} C_VEL
LIN {X 0,Y 467.569,Z 299.74,A -85,B 0,C 180,E1 -7530.665,E2 -7530.665} C_VEL
LIN {X 0,Y 467.606,Z 299.729,A -85,B 0,C 180,E1 -7533.2,E2 -7533.2} C_VEL
LIN {X 0,Y 467.582,Z 299.738,A -85,B 0,C 180,E1 -7536.468,E2 -7536.468} C_VEL
LIN {X 0,Y 467.613,Z 299.723,A -85,B 0,C 180,E1 -7539.777,E2 -7539.777} C_VEL
LIN {X 0,Y 467.599,Z 299.728,A -85,B 0,C 180,E1 -7542.507,E2 -7542.507} C_VEL
LIN {X 0,Y 467.597,Z 299.74,A -85,B 0,C 180,E1 -7545.197,E2 -7545.197} C_VEL
LIN {X 0,Y 467.647,Z 299.723,A -85,B 0,C 180,E1 -7547.855,E2 -7547.855} C_VEL
LIN {X 0,Y 467.672,Z 299.721,A -85,B 0,C 180,E1 -7551.358,E2 -7551.358} C_VEL
LIN {X 0,Y 467.733,Z 299.717,A -85,B 0,C 180,E1 -7553.963,E2 -7553.963} C_VEL
LIN {X 0,Y 467.85,Z 299.698,A -85,B 0,C 180,E1 -7557.418,E2 -7557.418} C_VEL
LIN {X 0,Y 467.871,Z 299.683,A -85,B 0,C 180,E1 -7560,E2 -7560} C_VEL
LIN {X 0,Y 467.85,Z 299.703,A -85,B 0,C 180,E1 -7562.583,E2 -7562.583} C_VEL
LIN {X 0,Y 467.734,Z 299.718,A -85,B 0,C 180,E1 -7566.038,E2 -7566.038} C_VEL
LIN {X 0,Y 467.673,Z 299.715,A -85,B 0,C 180,E1 -7568.643,E2 -7568.643} C_VEL
LIN {X 0,Y 467.648,Z 299.725,A -85,B 0,C 180,E1 -7572.146,E2 -7572.146} C_VEL
LIN {X 0,Y 467.631,Z 299.728,A -85,B 0,C 180,E1 -7575.696,E2 -7575.696} C_VEL
LIN {X 0,Y 467.609,Z 299.724,A -85,B 0,C 180,E1 -7578.765,E2 -7578.765} C_VEL
LIN {X 0,Y 467.572,Z 299.736,A -85,B 0,C 180,E1 -7581.269,E2 -7581.269} C_VEL
LIN {X 0,Y 467.554,Z 299.741,A -85,B 0,C 180,E1 -7583.945,E2 -7583.945} C_VEL
LIN {X 0,Y 467.606,Z 299.727,A -85,B 0,C 180,E1 -7586.801,E2 -7586.801} C_VEL
LIN {X 0,Y 467.547,Z 299.741,A -85,B 0,C 180,E1 -7589.739,E2 -7589.739} C_VEL
LIN {X 0,Y 467.567,Z 299.735,A -85,B 0,C 180,E1 -7592.76,E2 -7592.76} C_VEL
LIN {X 0,Y 467.547,Z 299.741,A -85,B 0,C 180,E1 -7595.891,E2 -7595.891} C_VEL
LIN {X 0,Y 467.555,Z 299.736,A -85,B 0,C 180,E1 -7599.148,E2 -7599.148} C_VEL
LIN {X 0,Y 467.583,Z 299.74,A -85,B 0,C 180,E1 -7602.568,E2 -7602.568} C_VEL
LIN {X 0,Y 467.562,Z 299.739,A -85,B 0,C 180,E1 -7605.053,E2 -7605.053} C_VEL
LIN {X 0,Y 467.571,Z 299.73,A -85,B 0,C 180,E1 -7608.598,E2 -7608.598} C_VEL
LIN {X 0,Y 467.56,Z 299.746,A -85,B 0,C 180,E1 -7611.956,E2 -7611.956} C_VEL
LIN {X 0,Y 467.561,Z 299.739,A -85,B 0,C 180,E1 -7615.168,E2 -7615.168} C_VEL
LIN {X 0,Y 467.582,Z 299.742,A -85,B 0,C 180,E1 -7618.261,E2 -7618.261} C_VEL
LIN {X 0,Y 467.576,Z 299.744,A -85,B 0,C 180,E1 -7621.251,E2 -7621.251} C_VEL
LIN {X 0,Y 467.695,Z 299.97,A -85,B 0,C 180,E1 -7622.5,E2 -7622.5} C_VEL
LIN {X 0,Y 469.43,Z 310.078,A -85,B 0,C 180,E1 -7624.98,E2 -7624.98} C_VEL
LIN {X 0,Y 469.001,Z 321.398,A -85,B 0,C 180,E1 -7627.536,E2 -7627.536} C_VEL
LIN {X 0,Y 468.305,Z 337.097,A -85,B 0,C 180,E1 -7630.991,E2 -7630.991} C_VEL
LIN {X 0,Y 467.949,Z 345.971,A -85,B 0,C 180,E1 -7632.942,E2 -7632.942} C_VEL
LIN {X 0,Y 468.452,Z 349.216,A -85,B 0,C 180,E1 -7633.059,E2 -7633.059} C_VEL
LIN {X 0,Y 471.218,Z 365.923,A -85,B 0,C 180,E1 -7633.421,E2 -7633.421} C_VEL
LIN {X 0,Y 470.58,Z 450.938,A -85,B 0,C 180,E1 -7634.739,E2 -7634.739} C_VEL
LIN {X 0,Y 470.305,Z 461.703,A -85,B 0,C 180,E1 -7635.007,E2 -7635.007} C_VEL
LIN {X 0,Y 470.046,Z 470.804,A -85,B 0,C 180,E1 -7635.331,E2 -7635.331} C_VEL
LIN {X 0,Y 469.608,Z 481.166,A -85,B 0,C 180,E1 -7635.815,E2 -7635.815} C_VEL
LIN {X 0,Y 469.24,Z 490.301,A -85,B 0,C 180,E1 -7636.356,E2 -7636.356} C_VEL
LIN {X 0,Y 468.828,Z 499.3,A -85,B 0,C 180,E1 -7637.006,E2 -7637.006} C_VEL
LIN {X 0,Y 468.52,Z 507.294,A -85,B 0,C 180,E1 -7637.696,E2 -7637.696} C_VEL
LIN {X 0,Y 468.129,Z 515.428,A -85,B 0,C 180,E1 -7638.526,E2 -7638.526} C_VEL
LIN {X 0,Y 467.744,Z 522.648,A -85,B 0,C 180,E1 -7639.394,E2 -7639.394} C_VEL
LIN {X 0,Y 467.464,Z 528.851,A -85,B 0,C 180,E1 -7640.263,E2 -7640.263} C_VEL
LIN {X 0,Y 467.164,Z 535.388,A -85,B 0,C 180,E1 -7641.348,E2 -7641.348} C_VEL
LIN {X 0,Y 466.991,Z 539.889,A -85,B 0,C 180,E1 -7642.216,E2 -7642.216} C_VEL
LIN {X 0,Y 466.797,Z 545.532,A -85,B 0,C 180,E1 -7643.56,E2 -7643.56} C_VEL
LIN {X 0,Y 466.738,Z 549.701,A -85,B 0,C 180,E1 -7644.817,E2 -7644.817} C_VEL
LIN {X 0,Y 466.649,Z 552.064,A -85,B 0,C 180,E1 -7645.681,E2 -7645.681} C_VEL
LIN {X 0,Y 466.689,Z 553.862,A -85,B 0,C 180,E1 -7646.547,E2 -7646.547} C_VEL
LIN {X 0,Y 466.608,Z 556.301,A -85,B 0,C 180,E1 -7648.274,E2 -7648.274} C_VEL
LIN {X 0,Y 466.619,Z 556.889,A -85,B 0,C 180,E1 -7649.137,E2 -7649.137} C_VEL
LIN {X 0,Y 466.619,Z 556.889,A -85,B 0,C 180,E1 -7650.863,E2 -7650.863} C_VEL
LIN {X 0,Y 466.608,Z 556.301,A -85,B 0,C 180,E1 -7651.726,E2 -7651.726} C_VEL
LIN {X 0,Y 466.689,Z 553.862,A -85,B 0,C 180,E1 -7653.453,E2 -7653.453} C_VEL
LIN {X 0,Y 466.692,Z 550.916,A -85,B 0,C 180,E1 -7654.751,E2 -7654.751} C_VEL
LIN {X 0,Y 466.749,Z 546.931,A -85,B 0,C 180,E1 -7656.05,E2 -7656.05} C_VEL
LIN {X 0,Y 466.935,Z 541.805,A -85,B 0,C 180,E1 -7657.35,E2 -7657.35} C_VEL
LIN {X 0,Y 467.118,Z 536.543,A -85,B 0,C 180,E1 -7658.435,E2 -7658.435} C_VEL
LIN {X 0,Y 467.383,Z 530.226,A -85,B 0,C 180,E1 -7659.521,E2 -7659.521} C_VEL
LIN {X 0,Y 467.625,Z 524.274,A -85,B 0,C 180,E1 -7660.39,E2 -7660.39} C_VEL
LIN {X 0,Y 468.02,Z 517.347,A -85,B 0,C 180,E1 -7661.257,E2 -7661.257} C_VEL
LIN {X 0,Y 468.403,Z 509.166,A -85,B 0,C 180,E1 -7662.125,E2 -7662.125} C_VEL
LIN {X 0,Y 468.742,Z 501.215,A -85,B 0,C 180,E1 -7662.841,E2 -7662.841} C_VEL
LIN {X 0,Y 469.201,Z 491.935,A -85,B 0,C 180,E1 -7663.535,E2 -7663.535} C_VEL
LIN {X 0,Y 469.61,Z 482.174,A -85,B 0,C 180,E1 -7664.13,E2 -7664.13} C_VEL
LIN {X 0,Y 469.962,Z 473.38,A -85,B 0,C 180,E1 -7664.561,E2 -7664.561} C_VEL
LIN {X 0,Y 470.286,Z 463.453,A -85,B 0,C 180,E1 -7664.938,E2 -7664.938} C_VEL
LIN {X 0,Y 470.543,Z 453.601,A -85,B 0,C 180,E1 -7665.207,E2 -7665.207} C_VEL
LIN {X 0,Y 470.809,Z 428.028,A -85,B 0,C 180,E1 -7665.629,E2 -7665.629} C_VEL
LIN {X 0,Y 471.084,Z 364.766,A -85,B 0,C 180,E1 -7666.602,E2 -7666.602} C_VEL
LIN {X 0,Y 467.996,Z 346.362,A -85,B 0,C 180,E1 -7667.021,E2 -7667.021} C_VEL
LIN {X 0,Y 467.969,Z 344.847,A -85,B 0,C 180,E1 -7667.276,E2 -7667.276} C_VEL
LIN {X 0,Y 468.614,Z 330.877,A -85,B 0,C 180,E1 -7670.407,E2 -7670.407} C_VEL
LIN {X 0,Y 469.228,Z 316.286,A -85,B 0,C 180,E1 -7673.619,E2 -7673.619} C_VEL
LIN {X 0,Y 469.416,Z 310.078,A -85,B 0,C 180,E1 -7675.021,E2 -7675.021} C_VEL
LIN {X 0,Y 467.682,Z 299.846,A -85,B 0,C 180,E1 -7677.549,E2 -7677.549} C_VEL
LIN {X 0,Y 467.568,Z 299.743,A -85,B 0,C 180,E1 -7681.044,E2 -7681.044} C_VEL
LIN {X 0,Y 467.587,Z 299.741,A -85,B 0,C 180,E1 -7684.241,E2 -7684.241} C_VEL
LIN {X 0,Y 467.541,Z 299.742,A -85,B 0,C 180,E1 -7687.184,E2 -7687.184} C_VEL
LIN {X 0,Y 467.568,Z 299.73,A -85,B 0,C 180,E1 -7690.264,E2 -7690.264} C_VEL
LIN {X 0,Y 467.547,Z 299.748,A -85,B 0,C 180,E1 -7693.744,E2 -7693.744} C_VEL
LIN {X 0,Y 467.547,Z 299.744,A -85,B 0,C 180,E1 -7696.254,E2 -7696.254} C_VEL
LIN {X 0,Y 467.574,Z 299.737,A -85,B 0,C 180,E1 -7698.722,E2 -7698.722} C_VEL
LIN {X 0,Y 467.56,Z 299.745,A -85,B 0,C 180,E1 -7701.954,E2 -7701.954} C_VEL
LIN {X 0,Y 467.552,Z 299.739,A -85,B 0,C 180,E1 -7705.166,E2 -7705.166} C_VEL
LIN {X 0,Y 467.572,Z 299.739,A -85,B 0,C 180,E1 -7708.259,E2 -7708.259} C_VEL
LIN {X 0,Y 467.57,Z 299.741,A -85,B 0,C 180,E1 -7711.25,E2 -7711.25} C_VEL
LIN {X 0,Y 467.59,Z 299.731,A -85,B 0,C 180,E1 -7714.158,E2 -7714.158} C_VEL
LIN {X 0,Y 467.568,Z 299.739,A -85,B 0,C 180,E1 -7716.995,E2 -7716.995} C_VEL
LIN {X 0,Y 467.616,Z 299.726,A -85,B 0,C 180,E1 -7719.776,E2 -7719.776} C_VEL
LIN {X 0,Y 467.6,Z 299.724,A -85,B 0,C 180,E1 -7722.506,E2 -7722.506} C_VEL
LIN {X 0,Y 467.601,Z 299.737,A -85,B 0,C 180,E1 -7725.196,E2 -7725.196} C_VEL
LIN {X 0,Y 467.648,Z 299.725,A -85,B 0,C 180,E1 -7727.854,E2 -7727.854} C_VEL
LIN {X 0,Y 467.673,Z 299.715,A -85,B 0,C 180,E1 -7731.357,E2 -7731.357} C_VEL
LIN {X 0,Y 467.734,Z 299.718,A -85,B 0,C 180,E1 -7733.962,E2 -7733.962} C_VEL
LIN {X 0,Y 467.85,Z 299.703,A -85,B 0,C 180,E1 -7737.417,E2 -7737.417} C_VEL
LIN {X 0,Y 467.871,Z 299.683,A -85,B 0,C 180,E1 -7740,E2 -7740} C_VEL
LIN {X 0,Y 467.85,Z 299.698,A -85,B 0,C 180,E1 -7742.582,E2 -7742.582} C_VEL
LIN {X 0,Y 467.733,Z 299.717,A -85,B 0,C 180,E1 -7746.037,E2 -7746.037} C_VEL
LIN {X 0,Y 467.672,Z 299.721,A -85,B 0,C 180,E1 -7748.642,E2 -7748.642} C_VEL
LIN {X 0,Y 467.647,Z 299.723,A -85,B 0,C 180,E1 -7752.145,E2 -7752.145} C_VEL
LIN {X 0,Y 467.628,Z 299.731,A -85,B 0,C 180,E1 -7755.695,E2 -7755.695} C_VEL
LIN {X 0,Y 467.607,Z 299.727,A -85,B 0,C 180,E1 -7758.764,E2 -7758.764} C_VEL
LIN {X 0,Y 467.57,Z 299.74,A -85,B 0,C 180,E1 -7761.268,E2 -7761.268} C_VEL
LIN {X 0,Y 467.562,Z 299.739,A -85,B 0,C 180,E1 -7763.943,E2 -7763.943} C_VEL
LIN {X 0,Y 467.606,Z 299.729,A -85,B 0,C 180,E1 -7766.8,E2 -7766.8} C_VEL
LIN {X 0,Y 467.578,Z 299.736,A -85,B 0,C 180,E1 -7769.736,E2 -7769.736} C_VEL
LIN {X 0,Y 467.574,Z 299.741,A -85,B 0,C 180,E1 -7772.758,E2 -7772.758} C_VEL
LIN {X 0,Y 467.547,Z 299.738,A -85,B 0,C 180,E1 -7775.889,E2 -7775.889} C_VEL
LIN {X 0,Y 467.606,Z 299.734,A -85,B 0,C 180,E1 -7779.142,E2 -7779.142} C_VEL
LIN {X 0,Y 467.611,Z 299.738,A -85,B 0,C 180,E1 -7782.572,E2 -7782.572} C_VEL
LIN {X 0,Y 467.559,Z 299.736,A -85,B 0,C 180,E1 -7786.178,E2 -7786.178} C_VEL
LIN {X 0,Y 467.574,Z 299.723,A -85,B 0,C 180,E1 -7788.723,E2 -7788.723} C_VEL
LIN {X 0,Y 467.559,Z 299.742,A -85,B 0,C 180,E1 -7791.956,E2 -7791.956} C_VEL
LIN {X 0,Y 467.561,Z 299.726,A -85,B 0,C 180,E1 -7795.168,E2 -7795.168} C_VEL
LIN {X 0,Y 467.578,Z 299.744,A -85,B 0,C 180,E1 -7798.26,E2 -7798.26} C_VEL
LIN {X 0,Y 467.571,Z 299.735,A -85,B 0,C 180,E1 -7801.251,E2 -7801.251} C_VEL
LIN {X 0,Y 467.606,Z 299.741,A -85,B 0,C 180,E1 -7804.161,E2 -7804.161} C_VEL
LIN {X 0,Y 467.573,Z 299.742,A -85,B 0,C 180,E1 -7806.996,E2 -7806.996} C_VEL
LIN {X 0,Y 467.618,Z 299.737,A -85,B 0,C 180,E1 -7809.777,E2 -7809.777} C_VEL
LIN {X 0,Y 467.605,Z 299.741,A -85,B 0,C 180,E1 -7812.507,E2 -7812.507} C_VEL
LIN {X 0,Y 467.592,Z 299.739,A -85,B 0,C 180,E1 -7815.434,E2 -7815.434} C_VEL
LIN {X 0,Y 466.923,Z 299.826,A -85,B 0,C 180,E1 -7816.153,E2 -7816.153} C_VEL
LIN {X 0,Y 464.079,Z 300.177,A -85,B 0,C 180,E1 -7817.322,E2 -7817.322} C_VEL
LIN {X 0,Y 461.68,Z 300.479,A -85,B 0,C 180,E1 -7818.264,E2 -7818.264} C_VEL
LIN {X 0,Y 460.655,Z 300.604,A -85,B 0,C 180,E1 -7818.991,E2 -7818.991} C_VEL
LIN {X 0,Y 460.573,Z 300.614,A -85,B 0,C 180,E1 -7819.238,E2 -7819.238} C_VEL
LIN {X 0,Y 460.716,Z 300.599,A -85,B 0,C 180,E1 -7822.538,E2 -7822.538} C_VEL
LIN {X 0,Y 460.694,Z 300.6,A -85,B 0,C 180,E1 -7824.748,E2 -7824.748} C_VEL
LIN {X 0,Y 460.822,Z 300.584,A -85,B 0,C 180,E1 -7827.378,E2 -7827.378} C_VEL
LIN {X 0,Y 460.85,Z 300.583,A -85,B 0,C 180,E1 -7830,E2 -7830} C_VEL
LIN {X 0,Y 460.822,Z 300.584,A -85,B 0,C 180,E1 -7832.622,E2 -7832.622} C_VEL
LIN {X 0,Y 460.707,Z 300.601,A -85,B 0,C 180,E1 -7836.13,E2 -7836.13} C_VEL
LIN {X 0,Y 460.625,Z 300.608,A -85,B 0,C 180,E1 -7838.776,E2 -7838.776} C_VEL
LIN {X 0,Y 460.609,Z 300.61,A -85,B 0,C 180,E1 -7842.445,E2 -7842.445} C_VEL
LIN {X 0,Y 460.596,Z 300.614,A -85,B 0,C 180,E1 -7845.997,E2 -7845.997} C_VEL
LIN {X 0,Y 460.566,Z 300.614,A -85,B 0,C 180,E1 -7848.902,E2 -7848.902} C_VEL
LIN {X 0,Y 460.511,Z 300.625,A -85,B 0,C 180,E1 -7851.485,E2 -7851.485} C_VEL
LIN {X 0,Y 460.538,Z 300.618,A -85,B 0,C 180,E1 -7854.332,E2 -7854.332} C_VEL
LIN {X 0,Y 460.578,Z 300.615,A -85,B 0,C 180,E1 -7857.243,E2 -7857.243} C_VEL
LIN {X 0,Y 460.505,Z 300.618,A -85,B 0,C 180,E1 -7860.24,E2 -7860.24} C_VEL
LIN {X 0,Y 460.523,Z 300.614,A -85,B 0,C 180,E1 -7863.324,E2 -7863.324} C_VEL
LIN {X 0,Y 460.472,Z 300.621,A -85,B 0,C 180,E1 -7866.529,E2 -7866.529} C_VEL
LIN {X 0,Y 460.559,Z 300.606,A -85,B 0,C 180,E1 -7869.858,E2 -7869.858} C_VEL
LIN {X 0,Y 460.508,Z 300.598,A -85,B 0,C 180,E1 -7872.901,E2 -7872.901} C_VEL
LIN {X 0,Y 460.511,Z 300.621,A -85,B 0,C 180,E1 -7875.829,E2 -7875.829} C_VEL
LIN {X 0,Y 460.534,Z 300.614,A -85,B 0,C 180,E1 -7878.99,E2 -7878.99} C_VEL
LIN {X 0,Y 460.535,Z 300.62,A -85,B 0,C 180,E1 -7881.269,E2 -7881.269} C_VEL
LIN {X 0,Y 460.504,Z 300.616,A -85,B 0,C 180,E1 -7884.555,E2 -7884.555} C_VEL
LIN {X 0,Y 460.523,Z 300.619,A -85,B 0,C 180,E1 -7887.716,E2 -7887.716} C_VEL
LIN {X 0,Y 460.538,Z 300.616,A -85,B 0,C 180,E1 -7890.77,E2 -7890.77} C_VEL
LIN {X 0,Y 460.553,Z 300.609,A -85,B 0,C 180,E1 -7893.735,E2 -7893.735} C_VEL
LIN {X 0,Y 460.536,Z 300.617,A -85,B 0,C 180,E1 -7896.624,E2 -7896.624} C_VEL
LIN {X 0,Y 460.542,Z 300.606,A -85,B 0,C 180,E1 -7899.453,E2 -7899.453} C_VEL
LIN {X 0,Y 460.549,Z 300.604,A -85,B 0,C 180,E1 -7902.23,E2 -7902.23} C_VEL
LIN {X 0,Y 460.555,Z 300.619,A -85,B 0,C 180,E1 -7904.965,E2 -7904.965} C_VEL
LIN {X 0,Y 460.599,Z 300.601,A -85,B 0,C 180,E1 -7907.666,E2 -7907.666} C_VEL
LIN {X 0,Y 460.619,Z 300.6,A -85,B 0,C 180,E1 -7911.224,E2 -7911.224} C_VEL
LIN {X 0,Y 460.699,Z 300.594,A -85,B 0,C 180,E1 -7913.87,E2 -7913.87} C_VEL
LIN {X 0,Y 460.791,Z 300.577,A -85,B 0,C 180,E1 -7917.378,E2 -7917.378} C_VEL
LIN {X 0,Y 460.842,Z 300.558,A -85,B 0,C 180,E1 -7920,E2 -7920} C_VEL
LIN {X 0,Y 460.815,Z 300.58,A -85,B 0,C 180,E1 -7922.623,E2 -7922.623} C_VEL
LIN {X 0,Y 460.7,Z 300.595,A -85,B 0,C 180,E1 -7926.131,E2 -7926.131} C_VEL
LIN {X 0,Y 460.62,Z 300.591,A -85,B 0,C 180,E1 -7928.777,E2 -7928.777} C_VEL
LIN {X 0,Y 460.605,Z 300.605,A -85,B 0,C 180,E1 -7932.446,E2 -7932.446} C_VEL
LIN {X 0,Y 460.592,Z 300.606,A -85,B 0,C 180,E1 -7935.998,E2 -7935.998} C_VEL
LIN {X 0,Y 460.563,Z 300.602,A -85,B 0,C 180,E1 -7938.902,E2 -7938.902} C_VEL
LIN {X 0,Y 460.508,Z 300.616,A -85,B 0,C 180,E1 -7941.486,E2 -7941.486} C_VEL
LIN {X 0,Y 460.522,Z 300.62,A -85,B 0,C 180,E1 -7944.334,E2 -7944.334} C_VEL
LIN {X 0,Y 460.564,Z 300.601,A -85,B 0,C 180,E1 -7947.245,E2 -7947.245} C_VEL
LIN {X 0,Y 460.504,Z 300.624,A -85,B 0,C 180,E1 -7950.241,E2 -7950.241} C_VEL
LIN {X 0,Y 460.51,Z 300.611,A -85,B 0,C 180,E1 -7953.327,E2 -7953.327} C_VEL
LIN {X 0,Y 460.471,Z 300.628,A -85,B 0,C 180,E1 -7956.53,E2 -7956.53} C_VEL
LIN {X 0,Y 460.521,Z 300.616,A -85,B 0,C 180,E1 -7959.864,E2 -7959.864} C_VEL
LIN {X 0,Y 460.508,Z 300.619,A -85,B 0,C 180,E1 -7962.901,E2 -7962.901} C_VEL
LIN {X 0,Y 460.504,Z 300.622,A -85,B 0,C 180,E1 -7965.832,E2 -7965.832} C_VEL
LIN {X 0,Y 460.525,Z 300.605,A -85,B 0,C 180,E1 -7968.989,E2 -7968.989} C_VEL
LIN {X 0,Y 460.497,Z 300.623,A -85,B 0,C 180,E1 -7972.377,E2 -7972.377} C_VEL
LIN {X 0,Y 460.545,Z 300.616,A -85,B 0,C 180,E1 -7975.625,E2 -7975.625} C_VEL
LIN {X 0,Y 460.537,Z 300.62,A -85,B 0,C 180,E1 -7978.745,E2 -7978.745} C_VEL
LIN {X 0,Y 460.625,Z 300.742,A -85,B 0,C 180,E1 -7982.244,E2 -7982.244} C_VEL
LIN {X 0,Y 462.439,Z 310.961,A -85,B 0,C 180,E1 -7984.816,E2 -7984.816} C_VEL
LIN {X 0,Y 462.166,Z 319.155,A -85,B 0,C 180,E1 -7986.711,E2 -7986.711} C_VEL
LIN {X 0,Y 461.536,Z 332.609,A -85,B 0,C 180,E1 -7989.732,E2 -7989.732} C_VEL
LIN {X 0,Y 460.954,Z 345.78,A -85,B 0,C 180,E1 -7992.675,E2 -7992.675} C_VEL
LIN {X 0,Y 461.544,Z 349.271,A -85,B 0,C 180,E1 -7992.802,E2 -7992.802} C_VEL
LIN {X 0,Y 464.402,Z 366.728,A -85,B 0,C 180,E1 -7993.186,E2 -7993.186} C_VEL
LIN {X 0,Y 463.752,Z 450.744,A -85,B 0,C 180,E1 -7994.509,E2 -7994.509} C_VEL
LIN {X 0,Y 463.461,Z 461.51,A -85,B 0,C 180,E1 -7994.78,E2 -7994.78} C_VEL
LIN {X 0,Y 463.188,Z 470.611,A -85,B 0,C 180,E1 -7995.109,E2 -7995.109} C_VEL
LIN {X 0,Y 462.733,Z 480.972,A -85,B 0,C 180,E1 -7995.6,E2 -7995.6} C_VEL
LIN {X 0,Y 462.349,Z 490.108,A -85,B 0,C 180,E1 -7996.149,E2 -7996.149} C_VEL
LIN {X 0,Y 461.894,Z 499.105,A -85,B 0,C 180,E1 -7996.807,E2 -7996.807} C_VEL
LIN {X 0,Y 461.538,Z 507.304,A -85,B 0,C 180,E1 -7997.527,E2 -7997.527} C_VEL
LIN {X 0,Y 461.127,Z 515.233,A -85,B 0,C 180,E1 -7998.35,E2 -7998.35} C_VEL
LIN {X 0,Y 460.734,Z 522.453,A -85,B 0,C 180,E1 -7999.231,E2 -7999.231} C_VEL
LIN {X 0,Y 460.448,Z 528.656,A -85,B 0,C 180,E1 -8000.113,E2 -8000.113} C_VEL
LIN {X 0,Y 460.125,Z 535.193,A -85,B 0,C 180,E1 -8001.214,E2 -8001.214} C_VEL
LIN {X 0,Y 459.935,Z 539.694,A -85,B 0,C 180,E1 -8002.096,E2 -8002.096} C_VEL
LIN {X 0,Y 459.743,Z 544.677,A -85,B 0,C 180,E1 -8003.273,E2 -8003.273} C_VEL
LIN {X 0,Y 459.651,Z 549.507,A -85,B 0,C 180,E1 -8004.736,E2 -8004.736} C_VEL
LIN {X 0,Y 459.566,Z 551.87,A -85,B 0,C 180,E1 -8005.615,E2 -8005.615} C_VEL
LIN {X 0,Y 459.584,Z 553.668,A -85,B 0,C 180,E1 -8006.493,E2 -8006.493} C_VEL
LIN {X 0,Y 459.521,Z 556.108,A -85,B 0,C 180,E1 -8008.247,E2 -8008.247} C_VEL
LIN {X 0,Y 459.522,Z 556.695,A -85,B 0,C 180,E1 -8009.124,E2 -8009.124} C_VEL
LIN {X 0,Y 459.522,Z 556.695,A -85,B 0,C 180,E1 -8010.876,E2 -8010.876} C_VEL
LIN {X 0,Y 459.521,Z 556.108,A -85,B 0,C 180,E1 -8011.753,E2 -8011.753} C_VEL
LIN {X 0,Y 459.584,Z 553.668,A -85,B 0,C 180,E1 -8013.507,E2 -8013.507} C_VEL
LIN {X 0,Y 459.619,Z 550.722,A -85,B 0,C 180,E1 -8014.824,E2 -8014.824} C_VEL
LIN {X 0,Y 459.66,Z 546.736,A -85,B 0,C 180,E1 -8016.144,E2 -8016.144} C_VEL
LIN {X 0,Y 459.856,Z 541.61,A -85,B 0,C 180,E1 -8017.464,E2 -8017.464} C_VEL
LIN {X 0,Y 460.052,Z 536.348,A -85,B 0,C 180,E1 -8018.566,E2 -8018.566} C_VEL
LIN {X 0,Y 460.366,Z 530.032,A -85,B 0,C 180,E1 -8019.667,E2 -8019.667} C_VEL
LIN {X 0,Y 460.609,Z 524.079,A -85,B 0,C 180,E1 -8020.55,E2 -8020.55} C_VEL
LIN {X 0,Y 461.035,Z 517.153,A -85,B 0,C 180,E1 -8021.43,E2 -8021.43} C_VEL
LIN {X 0,Y 461.444,Z 508.971,A -85,B 0,C 180,E1 -8022.311,E2 -8022.311} C_VEL
LIN {X 0,Y 461.828,Z 500.152,A -85,B 0,C 180,E1 -8023.108,E2 -8023.108} C_VEL
LIN {X 0,Y 462.274,Z 491.74,A -85,B 0,C 180,E1 -8023.742,E2 -8023.742} C_VEL
LIN {X 0,Y 462.719,Z 481.98,A -85,B 0,C 180,E1 -8024.345,E2 -8024.345} C_VEL
LIN {X 0,Y 463.1,Z 473.186,A -85,B 0,C 180,E1 -8024.782,E2 -8024.782} C_VEL
LIN {X 0,Y 463.434,Z 463.259,A -85,B 0,C 180,E1 -8025.164,E2 -8025.164} C_VEL
LIN {X 0,Y 463.714,Z 453.408,A -85,B 0,C 180,E1 -8025.436,E2 -8025.436} C_VEL
LIN {X 0,Y 463.96,Z 428,A -85,B 0,C 180,E1 -8025.863,E2 -8025.863} C_VEL
LIN {X 0,Y 464.299,Z 365.686,A -85,B 0,C 180,E1 -8026.834,E2 -8026.834} C_VEL
LIN {X 0,Y 460.972,Z 346.228,A -85,B 0,C 180,E1 -8027.285,E2 -8027.285} C_VEL
LIN {X 0,Y 460.964,Z 345.082,A -85,B 0,C 180,E1 -8027.444,E2 -8027.444} C_VEL
LIN {X 0,Y 461.612,Z 331.744,A -85,B 0,C 180,E1 -8030.497,E2 -8030.497} C_VEL
LIN {X 0,Y 462.21,Z 318.245,A -85,B 0,C 180,E1 -8033.524,E2 -8033.524} C_VEL
LIN {X 0,Y 462.419,Z 310.96,A -85,B 0,C 180,E1 -8035.185,E2 -8035.185} C_VEL
LIN {X 0,Y 460.619,Z 300.743,A -85,B 0,C 180,E1 -8037.754,E2 -8037.754} C_VEL
LIN {X 0,Y 460.521,Z 300.622,A -85,B 0,C 180,E1 -8041.282,E2 -8041.282} C_VEL
LIN {X 0,Y 460.53,Z 300.617,A -85,B 0,C 180,E1 -8044.504,E2 -8044.504} C_VEL
LIN {X 0,Y 460.497,Z 300.623,A -85,B 0,C 180,E1 -8047.623,E2 -8047.623} C_VEL
LIN {X 0,Y 460.525,Z 300.605,A -85,B 0,C 180,E1 -8051.011,E2 -8051.011} C_VEL
LIN {X 0,Y 460.51,Z 300.618,A -85,B 0,C 180,E1 -8054.588,E2 -8054.588} C_VEL
LIN {X 0,Y 460.519,Z 300.624,A -85,B 0,C 180,E1 -8057.818,E2 -8057.818} C_VEL
LIN {X 0,Y 460.529,Z 300.612,A -85,B 0,C 180,E1 -8061.103,E2 -8061.103} C_VEL
LIN {X 0,Y 460.503,Z 300.615,A -85,B 0,C 180,E1 -8064.553,E2 -8064.553} C_VEL
LIN {X 0,Y 460.519,Z 300.619,A -85,B 0,C 180,E1 -8067.714,E2 -8067.714} C_VEL
LIN {X 0,Y 460.533,Z 300.614,A -85,B 0,C 180,E1 -8070.768,E2 -8070.768} C_VEL
LIN {X 0,Y 460.549,Z 300.607,A -85,B 0,C 180,E1 -8073.733,E2 -8073.733} C_VEL
LIN {X 0,Y 460.536,Z 300.614,A -85,B 0,C 180,E1 -8076.623,E2 -8076.623} C_VEL
LIN {X 0,Y 460.544,Z 300.612,A -85,B 0,C 180,E1 -8079.452,E2 -8079.452} C_VEL
LIN {X 0,Y 460.551,Z 300.602,A -85,B 0,C 180,E1 -8082.229,E2 -8082.229} C_VEL
LIN {X 0,Y 460.559,Z 300.611,A -85,B 0,C 180,E1 -8084.964,E2 -8084.964} C_VEL
LIN {X 0,Y 460.604,Z 300.6,A -85,B 0,C 180,E1 -8088.559,E2 -8088.559} C_VEL
LIN {X 0,Y 460.686,Z 300.589,A -85,B 0,C 180,E1 -8092.108,E2 -8092.108} C_VEL
LIN {X 0,Y 460.688,Z 300.597,A -85,B 0,C 180,E1 -8094.748,E2 -8094.748} C_VEL
LIN {X 0,Y 460.815,Z 300.58,A -85,B 0,C 180,E1 -8097.377,E2 -8097.377} C_VEL
LIN {X 0,Y 460.842,Z 300.558,A -85,B 0,C 180,E1 -8100,E2 -8100} C_VEL
LIN {X 0,Y 460.791,Z 300.577,A -85,B 0,C 180,E1 -8102.622,E2 -8102.622} C_VEL
LIN {X 0,Y 460.699,Z 300.594,A -85,B 0,C 180,E1 -8106.13,E2 -8106.13} C_VEL
LIN {X 0,Y 460.619,Z 300.6,A -85,B 0,C 180,E1 -8108.776,E2 -8108.776} C_VEL
LIN {X 0,Y 460.603,Z 300.602,A -85,B 0,C 180,E1 -8112.445,E2 -8112.445} C_VEL
LIN {X 0,Y 460.59,Z 300.607,A -85,B 0,C 180,E1 -8115.997,E2 -8115.997} C_VEL
LIN {X 0,Y 460.56,Z 300.603,A -85,B 0,C 180,E1 -8118.902,E2 -8118.902} C_VEL
LIN {X 0,Y 460.505,Z 300.618,A -85,B 0,C 180,E1 -8121.486,E2 -8121.486} C_VEL
LIN {X 0,Y 460.532,Z 300.617,A -85,B 0,C 180,E1 -8124.332,E2 -8124.332} C_VEL
LIN {X 0,Y 460.563,Z 300.603,A -85,B 0,C 180,E1 -8127.244,E2 -8127.244} C_VEL
LIN {X 0,Y 460.518,Z 300.617,A -85,B 0,C 180,E1 -8130.239,E2 -8130.239} C_VEL
LIN {X 0,Y 460.52,Z 300.612,A -85,B 0,C 180,E1 -8133.325,E2 -8133.325} C_VEL
LIN {X 0,Y 460.47,Z 300.625,A -85,B 0,C 180,E1 -8136.529,E2 -8136.529} C_VEL
LIN {X 0,Y 460.567,Z 300.608,A -85,B 0,C 180,E1 -8139.858,E2 -8139.858} C_VEL
LIN {X 0,Y 460.532,Z 300.62,A -85,B 0,C 180,E1 -8142.904,E2 -8142.904} C_VEL
LIN {X 0,Y 460.511,Z 300.612,A -85,B 0,C 180,E1 -8145.83,E2 -8145.83} C_VEL
LIN {X 0,Y 460.527,Z 300.603,A -85,B 0,C 180,E1 -8148.989,E2 -8148.989} C_VEL
LIN {X 0,Y 460.523,Z 300.618,A -85,B 0,C 180,E1 -8151.268,E2 -8151.268} C_VEL
LIN {X 0,Y 460.507,Z 300.609,A -85,B 0,C 180,E1 -8154.555,E2 -8154.555} C_VEL
LIN {X 0,Y 460.526,Z 300.617,A -85,B 0,C 180,E1 -8157.716,E2 -8157.716} C_VEL
LIN {X 0,Y 460.534,Z 300.609,A -85,B 0,C 180,E1 -8160.769,E2 -8160.769} C_VEL
LIN {X 0,Y 460.563,Z 300.615,A -85,B 0,C 180,E1 -8163.735,E2 -8163.735} C_VEL
LIN {X 0,Y 460.541,Z 300.62,A -85,B 0,C 180,E1 -8166.624,E2 -8166.624} C_VEL
LIN {X 0,Y 460.547,Z 300.616,A -85,B 0,C 180,E1 -8169.453,E2 -8169.453} C_VEL
LIN {X 0,Y 460.555,Z 300.62,A -85,B 0,C 180,E1 -8172.23,E2 -8172.23} C_VEL
LIN {X 0,Y 460.561,Z 300.616,A -85,B 0,C 180,E1 -8174.965,E2 -8174.965} C_VEL
LIN {X 0,Y 460.608,Z 300.612,A -85,B 0,C 180,E1 -8178.559,E2 -8178.559} C_VEL
LIN {X 0,Y 460.573,Z 300.614,A -85,B 0,C 180,E1 -8179.238,E2 -8179.238} C_VEL
LIN {X 0,Y 459.92,Z 300.699,A -85,B 0,C 180,E1 -8179.968,E2 -8179.968} C_VEL
LIN {X 0,Y 457.102,Z 301.049,A -85,B 0,C 180,E1 -8181.155,E2 -8181.155} C_VEL
LIN {X 0,Y 454.722,Z 301.347,A -85,B 0,C 180,E1 -8182.112,E2 -8182.112} C_VEL
LIN {X 0,Y 453.711,Z 301.47,A -85,B 0,C 180,E1 -8182.851,E2 -8182.851} C_VEL
LIN {X 0,Y 453.634,Z 301.478,A -85,B 0,C 180,E1 -8183.101,E2 -8183.101} C_VEL
LIN {X 0,Y 453.668,Z 301.475,A -85,B 0,C 180,E1 -8184.667,E2 -8184.667} C_VEL
LIN {X 0,Y 453.762,Z 301.463,A -85,B 0,C 180,E1 -8187.337,E2 -8187.337} C_VEL
LIN {X 0,Y 453.821,Z 301.459,A -85,B 0,C 180,E1 -8190,E2 -8190} C_VEL
LIN {X 0,Y 453.762,Z 301.463,A -85,B 0,C 180,E1 -8192.663,E2 -8192.663} C_VEL
LIN {X 0,Y 453.674,Z 301.476,A -85,B 0,C 180,E1 -8196.225,E2 -8196.225} C_VEL
LIN {X 0,Y 453.589,Z 301.484,A -85,B 0,C 180,E1 -8198.913,E2 -8198.913} C_VEL
LIN {X 0,Y 453.559,Z 301.488,A -85,B 0,C 180,E1 -8202.529,E2 -8202.529} C_VEL
LIN {X 0,Y 453.54,Z 301.492,A -85,B 0,C 180,E1 -8206.196,E2 -8206.196} C_VEL
LIN {X 0,Y 453.516,Z 301.493,A -85,B 0,C 180,E1 -8209.041,E2 -8209.041} C_VEL
LIN {X 0,Y 453.472,Z 301.502,A -85,B 0,C 180,E1 -8211.836,E2 -8211.836} C_VEL
LIN {X 0,Y 453.509,Z 301.493,A -85,B 0,C 180,E1 -8214.734,E2 -8214.734} C_VEL
LIN {X 0,Y 453.532,Z 301.487,A -85,B 0,C 180,E1 -8217.961,E2 -8217.961} C_VEL
LIN {X 0,Y 453.461,Z 301.502,A -85,B 0,C 180,E1 -8221.525,E2 -8221.525} C_VEL
LIN {X 0,Y 453.482,Z 301.478,A -85,B 0,C 180,E1 -8224.777,E2 -8224.777} C_VEL
LIN {X 0,Y 453.468,Z 301.496,A -85,B 0,C 180,E1 -8228.31,E2 -8228.31} C_VEL
LIN {X 0,Y 453.507,Z 301.481,A -85,B 0,C 180,E1 -8230.606,E2 -8230.606} C_VEL
LIN {X 0,Y 453.465,Z 301.49,A -85,B 0,C 180,E1 -8234.22,E2 -8234.22} C_VEL
LIN {X 0,Y 453.481,Z 301.498,A -85,B 0,C 180,E1 -8237.008,E2 -8237.008} C_VEL
LIN {X 0,Y 453.522,Z 301.486,A -85,B 0,C 180,E1 -8240.554,E2 -8240.554} C_VEL
LIN {X 0,Y 453.448,Z 301.495,A -85,B 0,C 180,E1 -8243.917,E2 -8243.917} C_VEL
LIN {X 0,Y 453.474,Z 301.495,A -85,B 0,C 180,E1 -8247.151,E2 -8247.151} C_VEL
LIN {X 0,Y 453.505,Z 301.49,A -85,B 0,C 180,E1 -8250.271,E2 -8250.271} C_VEL
LIN {X 0,Y 453.496,Z 301.486,A -85,B 0,C 180,E1 -8253.294,E2 -8253.294} C_VEL
LIN {X 0,Y 453.493,Z 301.492,A -85,B 0,C 180,E1 -8256.239,E2 -8256.239} C_VEL
LIN {X 0,Y 453.473,Z 301.49,A -85,B 0,C 180,E1 -8259.118,E2 -8259.118} C_VEL
LIN {X 0,Y 453.501,Z 301.482,A -85,B 0,C 180,E1 -8261.945,E2 -8261.945} C_VEL
LIN {X 0,Y 453.53,Z 301.491,A -85,B 0,C 180,E1 -8264.727,E2 -8264.727} C_VEL
LIN {X 0,Y 453.553,Z 301.48,A -85,B 0,C 180,E1 -8267.471,E2 -8267.471} C_VEL
LIN {X 0,Y 453.583,Z 301.473,A -85,B 0,C 180,E1 -8271.087,E2 -8271.087} C_VEL
LIN {X 0,Y 453.667,Z 301.47,A -85,B 0,C 180,E1 -8273.775,E2 -8273.775} C_VEL
LIN {X 0,Y 453.735,Z 301.456,A -85,B 0,C 180,E1 -8277.337,E2 -8277.337} C_VEL
LIN {X 0,Y 453.812,Z 301.433,A -85,B 0,C 180,E1 -8280,E2 -8280} C_VEL
LIN {X 0,Y 453.755,Z 301.46,A -85,B 0,C 180,E1 -8282.664,E2 -8282.664} C_VEL
LIN {X 0,Y 453.668,Z 301.472,A -85,B 0,C 180,E1 -8286.226,E2 -8286.226} C_VEL
LIN {X 0,Y 453.584,Z 301.465,A -85,B 0,C 180,E1 -8288.914,E2 -8288.914} C_VEL
LIN {X 0,Y 453.555,Z 301.485,A -85,B 0,C 180,E1 -8292.53,E2 -8292.53} C_VEL
LIN {X 0,Y 453.537,Z 301.487,A -85,B 0,C 180,E1 -8296.197,E2 -8296.197} C_VEL
LIN {X 0,Y 453.512,Z 301.48,A -85,B 0,C 180,E1 -8299.041,E2 -8299.041} C_VEL
LIN {X 0,Y 453.469,Z 301.493,A -85,B 0,C 180,E1 -8301.837,E2 -8301.837} C_VEL
LIN {X 0,Y 453.492,Z 301.489,A -85,B 0,C 180,E1 -8304.736,E2 -8304.736} C_VEL
LIN {X 0,Y 453.526,Z 301.48,A -85,B 0,C 180,E1 -8307.96,E2 -8307.96} C_VEL
LIN {X 0,Y 453.457,Z 301.497,A -85,B 0,C 180,E1 -8311.525,E2 -8311.525} C_VEL
LIN {X 0,Y 453.476,Z 301.492,A -85,B 0,C 180,E1 -8314.777,E2 -8314.777} C_VEL
LIN {X 0,Y 453.455,Z 301.5,A -85,B 0,C 180,E1 -8318.313,E2 -8318.313} C_VEL
LIN {X 0,Y 453.49,Z 301.494,A -85,B 0,C 180,E1 -8320.61,E2 -8320.61} C_VEL
LIN {X 0,Y 453.449,Z 301.497,A -85,B 0,C 180,E1 -8323.245,E2 -8323.245} C_VEL
LIN {X 0,Y 453.459,Z 301.499,A -85,B 0,C 180,E1 -8325.779,E2 -8325.779} C_VEL
LIN {X 0,Y 453.491,Z 301.481,A -85,B 0,C 180,E1 -8329.41,E2 -8329.41} C_VEL
LIN {X 0,Y 453.448,Z 301.498,A -85,B 0,C 180,E1 -8332.811,E2 -8332.811} C_VEL
LIN {X 0,Y 453.476,Z 301.501,A -85,B 0,C 180,E1 -8336.088,E2 -8336.088} C_VEL
LIN {X 0,Y 453.476,Z 301.5,A -85,B 0,C 180,E1 -8339.241,E2 -8339.241} C_VEL
LIN {X 0,Y 453.571,Z 301.652,A -85,B 0,C 180,E1 -8342.032,E2 -8342.032} C_VEL
LIN {X 0,Y 455.406,Z 311.843,A -85,B 0,C 180,E1 -8344.644,E2 -8344.644} C_VEL
LIN {X 0,Y 455.351,Z 317.323,A -85,B 0,C 180,E1 -8345.954,E2 -8345.954} C_VEL
LIN {X 0,Y 454.618,Z 331.405,A -85,B 0,C 180,E1 -8349.173,E2 -8349.173} C_VEL
LIN {X 0,Y 454.038,Z 343.604,A -85,B 0,C 180,E1 -8351.967,E2 -8351.967} C_VEL
LIN {X 0,Y 453.952,Z 345.589,A -85,B 0,C 180,E1 -8352.399,E2 -8352.399} C_VEL
LIN {X 0,Y 454.473,Z 348.74,A -85,B 0,C 180,E1 -8352.52,E2 -8352.52} C_VEL
LIN {X 0,Y 457.606,Z 367.354,A -85,B 0,C 180,E1 -8352.942,E2 -8352.942} C_VEL
LIN {X 0,Y 456.911,Z 450.55,A -85,B 0,C 180,E1 -8354.271,E2 -8354.271} C_VEL
LIN {X 0,Y 456.581,Z 461.315,A -85,B 0,C 180,E1 -8354.545,E2 -8354.545} C_VEL
LIN {X 0,Y 456.323,Z 470.416,A -85,B 0,C 180,E1 -8354.879,E2 -8354.879} C_VEL
LIN {X 0,Y 455.848,Z 480.778,A -85,B 0,C 180,E1 -8355.377,E2 -8355.377} C_VEL
LIN {X 0,Y 455.444,Z 489.913,A -85,B 0,C 180,E1 -8355.934,E2 -8355.934} C_VEL
LIN {X 0,Y 454.975,Z 498.911,A -85,B 0,C 180,E1 -8356.603,E2 -8356.603} C_VEL
LIN {X 0,Y 454.571,Z 507.298,A -85,B 0,C 180,E1 -8357.352,E2 -8357.352} C_VEL
LIN {X 0,Y 454.152,Z 515.038,A -85,B 0,C 180,E1 -8358.168,E2 -8358.168} C_VEL
LIN {X 0,Y 453.703,Z 522.258,A -85,B 0,C 180,E1 -8359.062,E2 -8359.062} C_VEL
LIN {X 0,Y 453.421,Z 528.461,A -85,B 0,C 180,E1 -8359.958,E2 -8359.958} C_VEL
LIN {X 0,Y 453.052,Z 534.998,A -85,B 0,C 180,E1 -8361.076,E2 -8361.076} C_VEL
LIN {X 0,Y 452.881,Z 539.5,A -85,B 0,C 180,E1 -8361.972,E2 -8361.972} C_VEL
LIN {X 0,Y 452.647,Z 545.145,A -85,B 0,C 180,E1 -8363.358,E2 -8363.358} C_VEL
LIN {X 0,Y 452.565,Z 549.312,A -85,B 0,C 180,E1 -8364.654,E2 -8364.654} C_VEL
LIN {X 0,Y 452.488,Z 551.676,A -85,B 0,C 180,E1 -8365.546,E2 -8365.546} C_VEL
LIN {X 0,Y 452.481,Z 553.473,A -85,B 0,C 180,E1 -8366.438,E2 -8366.438} C_VEL
LIN {X 0,Y 452.437,Z 555.914,A -85,B 0,C 180,E1 -8368.22,E2 -8368.22} C_VEL
LIN {X 0,Y 452.429,Z 556.501,A -85,B 0,C 180,E1 -8369.11,E2 -8369.11} C_VEL
LIN {X 0,Y 452.429,Z 556.501,A -85,B 0,C 180,E1 -8370.89,E2 -8370.89} C_VEL
LIN {X 0,Y 452.437,Z 555.914,A -85,B 0,C 180,E1 -8371.78,E2 -8371.78} C_VEL
LIN {X 0,Y 452.481,Z 553.473,A -85,B 0,C 180,E1 -8373.562,E2 -8373.562} C_VEL
LIN {X 0,Y 452.547,Z 550.529,A -85,B 0,C 180,E1 -8374.9,E2 -8374.9} C_VEL
LIN {X 0,Y 452.585,Z 546.542,A -85,B 0,C 180,E1 -8376.24,E2 -8376.24} C_VEL
LIN {X 0,Y 452.789,Z 541.415,A -85,B 0,C 180,E1 -8377.581,E2 -8377.581} C_VEL
LIN {X 0,Y 453.011,Z 536.154,A -85,B 0,C 180,E1 -8378.7,E2 -8378.7} C_VEL
LIN {X 0,Y 453.338,Z 529.837,A -85,B 0,C 180,E1 -8379.818,E2 -8379.818} C_VEL
LIN {X 0,Y 453.601,Z 523.884,A -85,B 0,C 180,E1 -8380.715,E2 -8380.715} C_VEL
LIN {X 0,Y 454.05,Z 516.958,A -85,B 0,C 180,E1 -8381.608,E2 -8381.608} C_VEL
LIN {X 0,Y 454.489,Z 508.777,A -85,B 0,C 180,E1 -8382.503,E2 -8382.503} C_VEL
LIN {X 0,Y 454.866,Z 500.76,A -85,B 0,C 180,E1 -8383.245,E2 -8383.245} C_VEL
LIN {X 0,Y 455.358,Z 491.545,A -85,B 0,C 180,E1 -8383.954,E2 -8383.954} C_VEL
LIN {X 0,Y 455.828,Z 481.786,A -85,B 0,C 180,E1 -8384.566,E2 -8384.566} C_VEL
LIN {X 0,Y 456.228,Z 472.992,A -85,B 0,C 180,E1 -8385.01,E2 -8385.01} C_VEL
LIN {X 0,Y 456.588,Z 463.065,A -85,B 0,C 180,E1 -8385.397,E2 -8385.397} C_VEL
LIN {X 0,Y 456.89,Z 453.215,A -85,B 0,C 180,E1 -8385.673,E2 -8385.673} C_VEL
LIN {X 0,Y 457.141,Z 427.939,A -85,B 0,C 180,E1 -8386.104,E2 -8386.104} C_VEL
LIN {X 0,Y 457.509,Z 366.39,A -85,B 0,C 180,E1 -8387.077,E2 -8387.077} C_VEL
LIN {X 0,Y 453.981,Z 345.965,A -85,B 0,C 180,E1 -8387.564,E2 -8387.564} C_VEL
LIN {X 0,Y 453.986,Z 344.527,A -85,B 0,C 180,E1 -8387.81,E2 -8387.81} C_VEL
LIN {X 0,Y 454.653,Z 331.583,A -85,B 0,C 180,E1 -8390.826,E2 -8390.826} C_VEL
LIN {X 0,Y 455.383,Z 317.444,A -85,B 0,C 180,E1 -8394.051,E2 -8394.051} C_VEL
LIN {X 0,Y 455.4,Z 311.843,A -85,B 0,C 180,E1 -8395.356,E2 -8395.356} C_VEL
LIN {X 0,Y 453.571,Z 301.635,A -85,B 0,C 180,E1 -8397.968,E2 -8397.968} C_VEL
LIN {X 0,Y 453.466,Z 301.503,A -85,B 0,C 180,E1 -8401.524,E2 -8401.524} C_VEL
LIN {X 0,Y 453.486,Z 301.493,A -85,B 0,C 180,E1 -8404.776,E2 -8404.776} C_VEL
LIN {X 0,Y 453.456,Z 301.499,A -85,B 0,C 180,E1 -8408.311,E2 -8408.311} C_VEL
LIN {X 0,Y 453.491,Z 301.481,A -85,B 0,C 180,E1 -8410.608,E2 -8410.608} C_VEL
LIN {X 0,Y 453.459,Z 301.499,A -85,B 0,C 180,E1 -8414.221,E2 -8414.221} C_VEL
LIN {X 0,Y 453.457,Z 301.497,A -85,B 0,C 180,E1 -8417.004,E2 -8417.004} C_VEL
LIN {X 0,Y 453.49,Z 301.495,A -85,B 0,C 180,E1 -8419.408,E2 -8419.408} C_VEL
LIN {X 0,Y 453.444,Z 301.501,A -85,B 0,C 180,E1 -8422.226,E2 -8422.226} C_VEL
LIN {X 0,Y 453.476,Z 301.492,A -85,B 0,C 180,E1 -8425.223,E2 -8425.223} C_VEL
LIN {X 0,Y 453.457,Z 301.497,A -85,B 0,C 180,E1 -8428.475,E2 -8428.475} C_VEL
LIN {X 0,Y 453.526,Z 301.48,A -85,B 0,C 180,E1 -8432.04,E2 -8432.04} C_VEL
